LIN {X 0,Y 360.28,Z 379.159,A -85,B 0,C 180,E1 -13217.608,E2 -13217.608} C_VEL
LIN {X 0,Y 360.477,Z 375.778,A -85,B 0,C 180,E1 -13219.893,E2 -13219.893} C_VEL
LIN {X 0,Y 360.757,Z 372.266,A -85,B 0,C 180,E1 -13221.597,E2 -13221.597} C_VEL
LIN {X 0,Y 361.143,Z 367.827,A -85,B 0,C 180,E1 -13223.293,E2 -13223.293} C_VEL
LIN {X 0,Y 361.709,Z 361.416,A -85,B 0,C 180,E1 -13225.262,E2 -13225.262} C_VEL
LIN {X 0,Y 362.596,Z 353.445,A -85,B 0,C 180,E1 -13227.221,E2 -13227.221} C_VEL
LIN {X 0,Y 363.549,Z 345.118,A -85,B 0,C 180,E1 -13228.891,E2 -13228.891} C_VEL
LIN {X 0,Y 364.702,Z 335.103,A -85,B 0,C 180,E1 -13230.55,E2 -13230.55} C_VEL
LIN {X 0,Y 365.932,Z 324.301,A -85,B 0,C 180,E1 -13232.018,E2 -13232.018} C_VEL
LIN {X 0,Y 367.02,Z 312.884,A -85,B 0,C 180,E1 -13233.292,E2 -13233.292} C_VEL
LIN {X 0,Y 368.264,Z 300.783,A -85,B 0,C 180,E1 -13234.376,E2 -13234.376} C_VEL
LIN {X 0,Y 369.232,Z 287.496,A -85,B 0,C 180,E1 -13235.323,E2 -13235.323} C_VEL
LIN {X 0,Y 370.079,Z 273.64,A -85,B 0,C 180,E1 -13236.062,E2 -13236.062} C_VEL
LIN {X 0,Y 370.646,Z 259.224,A -85,B 0,C 180,E1 -13236.599,E2 -13236.599} C_VEL
LIN {X 0,Y 371.262,Z 235.703,A -85,B 0,C 180,E1 -13237.1,E2 -13237.1} C_VEL
LIN {X 0,Y 372.051,Z 196.143,A -85,B 0,C 180,E1 -13237.865,E2 -13237.865} C_VEL
LIN {X 0,Y 371.527,Z 190.322,A -85,B 0,C 180,E1 -13238.014,E2 -13238.014} C_VEL
LIN {X 0,Y 366.374,Z 171.636,A -85,B 0,C 180,E1 -13238.703,E2 -13238.703} C_VEL
LIN {X 0,Y 366.023,Z 165.818,A -85,B 0,C 180,E1 -13238.845,E2 -13238.845} C_VEL
LIN {X 0,Y 366.284,Z 150.787,A -85,B 0,C 180,E1 -13239.144,E2 -13239.144} C_VEL
LIN {X 0,Y 363.95,Z 139.954,A -85,B 0,C 180,E1 -13239.517,E2 -13239.517} C_VEL
LIN {X 0,Y 356.742,Z 120.401,A -85,B 0,C 180,E1 -13240.412,E2 -13240.412} C_VEL
LIN {X 0,Y 354.92,Z 111.908,A -85,B 0,C 180,E1 -13242.725,E2 -13242.725} C_VEL
LIN {X 0,Y 354.909,Z 111.899,A -85,B 0,C 180,E1 -13244.916,E2 -13244.916} C_VEL
LIN {X 0,Y 354.881,Z 111.901,A -85,B 0,C 180,E1 -13248.471,E2 -13248.471} C_VEL
LIN {X 0,Y 354.856,Z 111.905,A -85,B 0,C 180,E1 -13252.103,E2 -13252.103} C_VEL
LIN {X 0,Y 354.865,Z 111.905,A -85,B 0,C 180,E1 -13255.828,E2 -13255.828} C_VEL
LIN {X 0,Y 354.82,Z 111.911,A -85,B 0,C 180,E1 -13259.68,E2 -13259.68} C_VEL
LIN {X 0,Y 354.794,Z 111.913,A -85,B 0,C 180,E1 -13263.709,E2 -13263.709} C_VEL
LIN {X 0,Y 354.85,Z 111.906,A -85,B 0,C 180,E1 -13267.615,E2 -13267.615} C_VEL
LIN {X 0,Y 354.855,Z 111.907,A -85,B 0,C 180,E1 -13271.192,E2 -13271.192} C_VEL
LIN {X 0,Y 354.863,Z 111.907,A -85,B 0,C 180,E1 -13274.53,E2 -13274.53} C_VEL
LIN {X 0,Y 354.812,Z 111.91,A -85,B 0,C 180,E1 -13277.672,E2 -13277.672} C_VEL
LIN {X 0,Y 354.809,Z 111.915,A -85,B 0,C 180,E1 -13280.672,E2 -13280.672} C_VEL
LIN {X 0,Y 354.795,Z 111.916,A -85,B 0,C 180,E1 -13284.304,E2 -13284.304} C_VEL
LIN {X 0,Y 354.773,Z 111.915,A -85,B 0,C 180,E1 -13287.671,E2 -13287.671} C_VEL
LIN {X 0,Y 354.845,Z 111.908,A -85,B 0,C 180,E1 -13290.624,E2 -13290.624} C_VEL
LIN {X 0,Y 354.879,Z 111.907,A -85,B 0,C 180,E1 -13294.176,E2 -13294.176} C_VEL
LIN {X 0,Y 354.871,Z 111.907,A -85,B 0,C 180,E1 -13297.901,E2 -13297.901} C_VEL
LIN {X 0,Y 354.904,Z 111.904,A -85,B 0,C 180,E1 -13301.895,E2 -13301.895} C_VEL
LIN {X 0,Y 354.926,Z 111.9,A -85,B 0,C 180,E1 -13305.984,E2 -13305.984} C_VEL
LIN {X 0,Y 354.967,Z 111.896,A -85,B 0,C 180,E1 -13309.74,E2 -13309.74} C_VEL
LIN {X 0,Y 355.1,Z 111.875,A -85,B 0,C 180,E1 -13312.041,E2 -13312.041} C_VEL
LIN {X 0,Y 355.081,Z 111.876,A -85,B 0,C 180,E1 -13314.324,E2 -13314.324} C_VEL
LIN {X 0,Y 355.235,Z 111.86,A -85,B 0,C 180,E1 -13317.736,E2 -13317.736} C_VEL
LIN {X 0,Y 355.388,Z 111.839,A -85,B 0,C 180,E1 -13320.004,E2 -13320.004} C_VEL
LIN {X 0,Y 355.236,Z 111.857,A -85,B 0,C 180,E1 -13322.271,E2 -13322.271} C_VEL
LIN {X 0,Y 355.13,Z 111.873,A -85,B 0,C 180,E1 -13326.823,E2 -13326.823} C_VEL
LIN {X 0,Y 355.007,Z 111.891,A -85,B 0,C 180,E1 -13329.116,E2 -13329.116} C_VEL
LIN {X 0,Y 354.914,Z 111.899,A -85,B 0,C 180,E1 -13332.584,E2 -13332.584} C_VEL
LIN {X 0,Y 354.884,Z 111.901,A -85,B 0,C 180,E1 -13336.1,E2 -13336.1} C_VEL
LIN {X 0,Y 354.902,Z 111.902,A -85,B 0,C 180,E1 -13338.475,E2 -13338.475} C_VEL
LIN {X 0,Y 354.831,Z 111.909,A -85,B 0,C 180,E1 -13342.109,E2 -13342.109} C_VEL
LIN {X 0,Y 354.897,Z 111.9,A -85,B 0,C 180,E1 -13345.831,E2 -13345.831} C_VEL
LIN {X 0,Y 354.852,Z 111.905,A -85,B 0,C 180,E1 -13349.682,E2 -13349.682} C_VEL
LIN {X 0,Y 354.805,Z 111.912,A -85,B 0,C 180,E1 -13353.705,E2 -13353.705} C_VEL
LIN {X 0,Y 354.798,Z 111.915,A -85,B 0,C 180,E1 -13356.463,E2 -13356.463} C_VEL
LIN {X 0,Y 354.825,Z 111.909,A -85,B 0,C 180,E1 -13359.427,E2 -13359.427} C_VEL
LIN {X 0,Y 354.789,Z 111.913,A -85,B 0,C 180,E1 -13362.87,E2 -13362.87} C_VEL
LIN {X 0,Y 354.769,Z 111.919,A -85,B 0,C 180,E1 -13366.106,E2 -13366.106} C_VEL
LIN {X 0,Y 354.789,Z 111.913,A -85,B 0,C 180,E1 -13369.182,E2 -13369.182} C_VEL
LIN {X 0,Y 354.809,Z 111.911,A -85,B 0,C 180,E1 -13372.406,E2 -13372.406} C_VEL
LIN {X 0,Y 354.815,Z 111.91,A -85,B 0,C 180,E1 -13374.943,E2 -13374.943} C_VEL
LIN {X 0,Y 354.842,Z 111.993,A -85,B 0,C 180,E1 -13377.708,E2 -13377.708} C_VEL
LIN {X 0,Y 357.811,Z 125.266,A -85,B 0,C 180,E1 -13380.916,E2 -13380.916} C_VEL
LIN {X 0,Y 359.778,Z 135.593,A -85,B 0,C 180,E1 -13383.304,E2 -13383.304} C_VEL
LIN {X 0,Y 359.646,Z 137.884,A -85,B 0,C 180,E1 -13383.792,E2 -13383.792} C_VEL
LIN {X 0,Y 365.98,Z 177.278,A -85,B 0,C 180,E1 -13385.03,E2 -13385.03} C_VEL
LIN {X 0,Y 363.987,Z 275.483,A -85,B 0,C 180,E1 -13386.985,E2 -13386.985} C_VEL
LIN {X 0,Y 363.267,Z 289.582,A -85,B 0,C 180,E1 -13387.463,E2 -13387.463} C_VEL
LIN {X 0,Y 362.303,Z 303.328,A -85,B 0,C 180,E1 -13388.15,E2 -13388.15} C_VEL
LIN {X 0,Y 361.223,Z 315.883,A -85,B 0,C 180,E1 -13388.988,E2 -13388.988} C_VEL
LIN {X 0,Y 360.036,Z 328.122,A -85,B 0,C 180,E1 -13390.027,E2 -13390.027} C_VEL
LIN {X 0,Y 358.739,Z 340.084,A -85,B 0,C 180,E1 -13391.291,E2 -13391.291} C_VEL
LIN {X 0,Y 357.568,Z 350.013,A -85,B 0,C 180,E1 -13392.56,E2 -13392.56} C_VEL
LIN {X 0,Y 356.484,Z 359.316,A -85,B 0,C 180,E1 -13393.98,E2 -13393.98} C_VEL
LIN {X 0,Y 355.424,Z 369.309,A -85,B 0,C 180,E1 -13395.837,E2 -13395.837} C_VEL
LIN {X 0,Y 354.616,Z 377.497,A -85,B 0,C 180,E1 -13397.701,E2 -13397.701} C_VEL
LIN {X 0,Y 353.863,Z 384.642,A -85,B 0,C 180,E1 -13399.705,E2 -13399.705} C_VEL
LIN {X 0,Y 353.574,Z 389.609,A -85,B 0,C 180,E1 -13401.428,E2 -13401.428} C_VEL
LIN {X 0,Y 353.325,Z 393.615,A -85,B 0,C 180,E1 -13403.147,E2 -13403.147} C_VEL
LIN {X 0,Y 353.231,Z 397.552,A -85,B 0,C 180,E1 -13405.437,E2 -13405.437} C_VEL
LIN {X 0,Y 353.173,Z 400.031,A -85,B 0,C 180,E1 -13407.721,E2 -13407.721} C_VEL
LIN {X 0,Y 353.266,Z 401.147,A -85,B 0,C 180,E1 -13410.002,E2 -13410.002} C_VEL
LIN {X 0,Y 353.169,Z 400.916,A -85,B 0,C 180,E1 -13412.283,E2 -13412.283} C_VEL
LIN {X 0,Y 353.24,Z 399.355,A -85,B 0,C 180,E1 -13414.566,E2 -13414.566} C_VEL
LIN {X 0,Y 353.403,Z 396.435,A -85,B 0,C 180,E1 -13416.854,E2 -13416.854} C_VEL
LIN {X 0,Y 353.783,Z 392.087,A -85,B 0,C 180,E1 -13419.146,E2 -13419.146} C_VEL
LIN {X 0,Y 354.433,Z 386.192,A -85,B 0,C 180,E1 -13421.438,E2 -13421.438} C_VEL
LIN {X 0,Y 355.535,Z 379.584,A -85,B 0,C 180,E1 -13423.432,E2 -13423.432} C_VEL
LIN {X 0,Y 356.689,Z 371.416,A -85,B 0,C 180,E1 -13425.427,E2 -13425.427} C_VEL
LIN {X 0,Y 358.106,Z 362.903,A -85,B 0,C 180,E1 -13427.122,E2 -13427.122} C_VEL
LIN {X 0,Y 359.813,Z 352.629,A -85,B 0,C 180,E1 -13428.803,E2 -13428.803} C_VEL
LIN {X 0,Y 361.692,Z 341.173,A -85,B 0,C 180,E1 -13430.325,E2 -13430.325} C_VEL
LIN {X 0,Y 363.54,Z 328.705,A -85,B 0,C 180,E1 -13431.666,E2 -13431.666} C_VEL
LIN {X 0,Y 365.24,Z 315.605,A -85,B 0,C 180,E1 -13432.785,E2 -13432.785} C_VEL
LIN {X 0,Y 366.662,Z 302.384,A -85,B 0,C 180,E1 -13433.662,E2 -13433.662} C_VEL
LIN {X 0,Y 368.012,Z 287.946,A -85,B 0,C 180,E1 -13434.356,E2 -13434.356} C_VEL
LIN {X 0,Y 368.924,Z 273.358,A -85,B 0,C 180,E1 -13434.817,E2 -13434.817} C_VEL
LIN {X 0,Y 371.332,Z 177.638,A -85,B 0,C 180,E1 -13436.751,E2 -13436.751} C_VEL
LIN {X 0,Y 366.862,Z 154.52,A -85,B 0,C 180,E1 -13437.693,E2 -13437.693} C_VEL
LIN {X 0,Y 364.291,Z 144.347,A -85,B 0,C 180,E1 -13438.178,E2 -13438.178} C_VEL
LIN {X 0,Y 361.13,Z 137.187,A -85,B 0,C 180,E1 -13438.682,E2 -13438.682} C_VEL
LIN {X 0,Y 358.951,Z 127.411,A -85,B 0,C 180,E1 -13441.256,E2 -13441.256} C_VEL
LIN {X 0,Y 356.041,Z 116.351,A -85,B 0,C 180,E1 -13444.371,E2 -13444.371} C_VEL
LIN {X 0,Y 354.85,Z 111.912,A -85,B 0,C 180,E1 -13445.702,E2 -13445.702} C_VEL
LIN {X 0,Y 354.814,Z 111.911,A -85,B 0,C 180,E1 -13449.418,E2 -13449.418} C_VEL
LIN {X 0,Y 354.801,Z 111.913,A -85,B 0,C 180,E1 -13452.866,E2 -13452.866} C_VEL
LIN {X 0,Y 354.782,Z 111.92,A -85,B 0,C 180,E1 -13456.103,E2 -13456.103} C_VEL
LIN {X 0,Y 354.797,Z 111.895,A -85,B 0,C 180,E1 -13459.177,E2 -13459.177} C_VEL
LIN {X 0,Y 354.815,Z 111.908,A -85,B 0,C 180,E1 -13462.403,E2 -13462.403} C_VEL
LIN {X 0,Y 354.823,Z 111.911,A -85,B 0,C 180,E1 -13464.939,E2 -13464.939} C_VEL
LIN {X 0,Y 354.808,Z 111.909,A -85,B 0,C 180,E1 -13468.404,E2 -13468.404} C_VEL
LIN {X 0,Y 354.817,Z 111.907,A -85,B 0,C 180,E1 -13471.613,E2 -13471.613} C_VEL
LIN {X 0,Y 354.865,Z 111.899,A -85,B 0,C 180,E1 -13475.421,E2 -13475.421} C_VEL
LIN {X 0,Y 354.841,Z 111.903,A -85,B 0,C 180,E1 -13479.111,E2 -13479.111} C_VEL
LIN {X 0,Y 354.912,Z 111.899,A -85,B 0,C 180,E1 -13482.717,E2 -13482.717} C_VEL
LIN {X 0,Y 354.964,Z 111.895,A -85,B 0,C 180,E1 -13486.252,E2 -13486.252} C_VEL
LIN {X 0,Y 354.967,Z 111.891,A -85,B 0,C 180,E1 -13489.732,E2 -13489.732} C_VEL
LIN {X 0,Y 355.099,Z 111.872,A -85,B 0,C 180,E1 -13493.177,E2 -13493.177} C_VEL
LIN {X 0,Y 355.242,Z 111.852,A -85,B 0,C 180,E1 -13497.729,E2 -13497.729} C_VEL
LIN {X 0,Y 355.36,Z 111.843,A -85,B 0,C 180,E1 -13499.996,E2 -13499.996} C_VEL
LIN {X 0,Y 355.247,Z 111.856,A -85,B 0,C 180,E1 -13502.264,E2 -13502.264} C_VEL
LIN {X 0,Y 355.104,Z 111.875,A -85,B 0,C 180,E1 -13506.816,E2 -13506.816} C_VEL
LIN {X 0,Y 354.959,Z 111.892,A -85,B 0,C 180,E1 -13510.26,E2 -13510.26} C_VEL
LIN {X 0,Y 354.945,Z 111.894,A -85,B 0,C 180,E1 -13514.014,E2 -13514.014} C_VEL
LIN {X 0,Y 354.922,Z 111.899,A -85,B 0,C 180,E1 -13518.104,E2 -13518.104} C_VEL
LIN {X 0,Y 354.827,Z 111.91,A -85,B 0,C 180,E1 -13522.102,E2 -13522.102} C_VEL
LIN {X 0,Y 354.892,Z 111.898,A -85,B 0,C 180,E1 -13525.823,E2 -13525.823} C_VEL
LIN {X 0,Y 354.8,Z 111.896,A -85,B 0,C 180,E1 -13529.678,E2 -13529.678} C_VEL
LIN {X 0,Y 354.804,Z 111.903,A -85,B 0,C 180,E1 -13533.679,E2 -13533.679} C_VEL
LIN {X 0,Y 354.786,Z 111.919,A -85,B 0,C 180,E1 -13536.455,E2 -13536.455} C_VEL
LIN {X 0,Y 354.811,Z 111.916,A -85,B 0,C 180,E1 -13539.419,E2 -13539.419} C_VEL
LIN {X 0,Y 354.779,Z 112.029,A -85,B 0,C 180,E1 -13542.094,E2 -13542.094} C_VEL
LIN {X 0,Y 357.266,Z 121.425,A -85,B 0,C 180,E1 -13544.98,E2 -13544.98} C_VEL
LIN {X 0,Y 367.344,Z 141.773,A -85,B 0,C 180,E1 -13546.486,E2 -13546.486} C_VEL
LIN {X 0,Y 371.616,Z 152.058,A -85,B 0,C 180,E1 -13547.126,E2 -13547.126} C_VEL
LIN {X 0,Y 371.984,Z 155.184,A -85,B 0,C 180,E1 -13547.23,E2 -13547.23} C_VEL
LIN {X 0,Y 369.169,Z 257.932,A -85,B 0,C 180,E1 -13549.303,E2 -13549.303} C_VEL
LIN {X 0,Y 368.327,Z 272.35,A -85,B 0,C 180,E1 -13549.815,E2 -13549.815} C_VEL
LIN {X 0,Y 367.121,Z 286.785,A -85,B 0,C 180,E1 -13550.569,E2 -13550.569} C_VEL
LIN {X 0,Y 365.711,Z 300.307,A -85,B 0,C 180,E1 -13551.524,E2 -13551.524} C_VEL
LIN {X 0,Y 364.152,Z 312.611,A -85,B 0,C 180,E1 -13552.634,E2 -13552.634} C_VEL
LIN {X 0,Y 362.478,Z 324.097,A -85,B 0,C 180,E1 -13553.917,E2 -13553.917} C_VEL
LIN {X 0,Y 360.851,Z 334.55,A -85,B 0,C 180,E1 -13555.345,E2 -13555.345} C_VEL
LIN {X 0,Y 359.349,Z 343.369,A -85,B 0,C 180,E1 -13556.795,E2 -13556.795} C_VEL
LIN {X 0,Y 357.753,Z 352.616,A -85,B 0,C 180,E1 -13558.627,E2 -13558.627} C_VEL
LIN {X 0,Y 356.399,Z 360.167,A -85,B 0,C 180,E1 -13560.461,E2 -13560.461} C_VEL
LIN {X 0,Y 355.416,Z 366.333,A -85,B 0,C 180,E1 -13562.308,E2 -13562.308} C_VEL
LIN {X 0,Y 354.591,Z 371.3,A -85,B 0,C 180,E1 -13564.147,E2 -13564.147} C_VEL
LIN {X 0,Y 354.04,Z 375.121,A -85,B 0,C 180,E1 -13565.929,E2 -13565.929} C_VEL
LIN {X 0,Y 353.596,Z 378.199,A -85,B 0,C 180,E1 -13567.811,E2 -13567.811} C_VEL
LIN {X 0,Y 353.224,Z 380.722,A -85,B 0,C 180,E1 -13570.228,E2 -13570.228} C_VEL
LIN {X 0,Y 353.081,Z 381.77,A -85,B 0,C 180,E1 -13572.627,E2 -13572.627} C_VEL
LIN {X 0,Y 353.002,Z 381.395,A -85,B 0,C 180,E1 -13574.998,E2 -13574.998} C_VEL
LIN {X 0,Y 353.166,Z 379.613,A -85,B 0,C 180,E1 -13577.354,E2 -13577.354} C_VEL
LIN {X 0,Y 353.349,Z 376.424,A -85,B 0,C 180,E1 -13579.686,E2 -13579.686} C_VEL
LIN {X 0,Y 353.639,Z 373.009,A -85,B 0,C 180,E1 -13581.427,E2 -13581.427} C_VEL
LIN {X 0,Y 354.195,Z 367.1,A -85,B 0,C 180,E1 -13583.733,E2 -13583.733} C_VEL
LIN {X 0,Y 354.834,Z 360.46,A -85,B 0,C 180,E1 -13585.739,E2 -13585.739} C_VEL
LIN {X 0,Y 355.776,Z 352.193,A -85,B 0,C 180,E1 -13587.734,E2 -13587.734} C_VEL
LIN {X 0,Y 356.804,Z 343.568,A -85,B 0,C 180,E1 -13589.434,E2 -13589.434} C_VEL
LIN {X 0,Y 358.02,Z 333.131,A -85,B 0,C 180,E1 -13591.123,E2 -13591.123} C_VEL
LIN {X 0,Y 359.353,Z 321.46,A -85,B 0,C 180,E1 -13592.661,E2 -13592.661} C_VEL
LIN {X 0,Y 360.595,Z 309.782,A -85,B 0,C 180,E1 -13593.91,E2 -13593.91} C_VEL
LIN {X 0,Y 361.772,Z 296.951,A -85,B 0,C 180,E1 -13595.014,E2 -13595.014} C_VEL
LIN {X 0,Y 362.808,Z 283.611,A -85,B 0,C 180,E1 -13595.905,E2 -13595.905} C_VEL
LIN {X 0,Y 363.558,Z 269.855,A -85,B 0,C 180,E1 -13596.589,E2 -13596.589} C_VEL
LIN {X 0,Y 364.059,Z 255.517,A -85,B 0,C 180,E1 -13597.067,E2 -13597.067} C_VEL
LIN {X 0,Y 366.023,Z 165.818,A -85,B 0,C 180,E1 -13598.845,E2 -13598.845} C_VEL
LIN {X 0,Y 365.619,Z 159.993,A -85,B 0,C 180,E1 -13598.992,E2 -13598.992} C_VEL
LIN {X 0,Y 364.039,Z 154.409,A -85,B 0,C 180,E1 -13599.207,E2 -13599.207} C_VEL
LIN {X 0,Y 359.047,Z 143.816,A -85,B 0,C 180,E1 -13599.745,E2 -13599.745} C_VEL
LIN {X 0,Y 355.643,Z 136.727,A -85,B 0,C 180,E1 -13600.119,E2 -13600.119} C_VEL
LIN {X 0,Y 349.585,Z 120.631,A -85,B 0,C 180,E1 -13600.89,E2 -13600.89} C_VEL
LIN {X 0,Y 347.909,Z 112.78,A -85,B 0,C 180,E1 -13603.06,E2 -13603.06} C_VEL
LIN {X 0,Y 347.824,Z 112.782,A -85,B 0,C 180,E1 -13606.43,E2 -13606.43} C_VEL
LIN {X 0,Y 347.831,Z 112.781,A -85,B 0,C 180,E1 -13608.86,E2 -13608.86} C_VEL
LIN {X 0,Y 347.776,Z 112.787,A -85,B 0,C 180,E1 -13612.577,E2 -13612.577} C_VEL
LIN {X 0,Y 347.786,Z 112.789,A -85,B 0,C 180,E1 -13615.108,E2 -13615.108} C_VEL
LIN {X 0,Y 347.777,Z 112.788,A -85,B 0,C 180,E1 -13617.695,E2 -13617.695} C_VEL
LIN {X 0,Y 347.736,Z 112.791,A -85,B 0,C 180,E1 -13620.347,E2 -13620.347} C_VEL
LIN {X 0,Y 347.731,Z 112.792,A -85,B 0,C 180,E1 -13624.049,E2 -13624.049} C_VEL
LIN {X 0,Y 347.794,Z 112.787,A -85,B 0,C 180,E1 -13627.314,E2 -13627.314} C_VEL
LIN {X 0,Y 347.787,Z 112.786,A -85,B 0,C 180,E1 -13630.287,E2 -13630.287} C_VEL
LIN {X 0,Y 347.79,Z 112.784,A -85,B 0,C 180,E1 -13633.395,E2 -13633.395} C_VEL
LIN {X 0,Y 347.789,Z 112.79,A -85,B 0,C 180,E1 -13636.672,E2 -13636.672} C_VEL
LIN {X 0,Y 347.757,Z 112.79,A -85,B 0,C 180,E1 -13640.168,E2 -13640.168} C_VEL
LIN {X 0,Y 347.763,Z 112.79,A -85,B 0,C 180,E1 -13644.128,E2 -13644.128} C_VEL
LIN {X 0,Y 347.74,Z 112.796,A -85,B 0,C 180,E1 -13648.306,E2 -13648.306} C_VEL
LIN {X 0,Y 347.783,Z 112.784,A -85,B 0,C 180,E1 -13650.993,E2 -13650.993} C_VEL
LIN {X 0,Y 347.81,Z 112.782,A -85,B 0,C 180,E1 -13653.611,E2 -13653.611} C_VEL
LIN {X 0,Y 347.797,Z 112.789,A -85,B 0,C 180,E1 -13656.168,E2 -13656.168} C_VEL
LIN {X 0,Y 347.825,Z 112.785,A -85,B 0,C 180,E1 -13659.915,E2 -13659.915} C_VEL
LIN {X 0,Y 347.849,Z 112.779,A -85,B 0,C 180,E1 -13662.363,E2 -13662.363} C_VEL
LIN {X 0,Y 347.88,Z 112.777,A -85,B 0,C 180,E1 -13665.975,E2 -13665.975} C_VEL
LIN {X 0,Y 347.918,Z 112.773,A -85,B 0,C 180,E1 -13669.53,E2 -13669.53} C_VEL
LIN {X 0,Y 348.06,Z 112.753,A -85,B 0,C 180,E1 -13671.879,E2 -13671.879} C_VEL
LIN {X 0,Y 348.056,Z 112.75,A -85,B 0,C 180,E1 -13674.21,E2 -13674.21} C_VEL
LIN {X 0,Y 348.198,Z 112.737,A -85,B 0,C 180,E1 -13677.69,E2 -13677.69} C_VEL
LIN {X 0,Y 348.358,Z 112.714,A -85,B 0,C 180,E1 -13680.004,E2 -13680.004} C_VEL
LIN {X 0,Y 348.199,Z 112.733,A -85,B 0,C 180,E1 -13682.317,E2 -13682.317} C_VEL
LIN {X 0,Y 348.098,Z 112.749,A -85,B 0,C 180,E1 -13686.961,E2 -13686.961} C_VEL
LIN {X 0,Y 347.96,Z 112.767,A -85,B 0,C 180,E1 -13689.302,E2 -13689.302} C_VEL
LIN {X 0,Y 347.883,Z 112.778,A -85,B 0,C 180,E1 -13692.843,E2 -13692.843} C_VEL
LIN {X 0,Y 347.834,Z 112.781,A -85,B 0,C 180,E1 -13696.435,E2 -13696.435} C_VEL
LIN {X 0,Y 347.851,Z 112.782,A -85,B 0,C 180,E1 -13698.864,E2 -13698.864} C_VEL
LIN {X 0,Y 347.771,Z 112.792,A -85,B 0,C 180,E1 -13702.583,E2 -13702.583} C_VEL
LIN {X 0,Y 347.809,Z 112.783,A -85,B 0,C 180,E1 -13705.112,E2 -13705.112} C_VEL
LIN {X 0,Y 347.809,Z 112.782,A -85,B 0,C 180,E1 -13707.697,E2 -13707.697} C_VEL
LIN {X 0,Y 347.762,Z 112.793,A -85,B 0,C 180,E1 -13710.35,E2 -13710.35} C_VEL
LIN {X 0,Y 347.744,Z 112.794,A -85,B 0,C 180,E1 -13714.467,E2 -13714.467} C_VEL
LIN {X 0,Y 347.773,Z 112.791,A -85,B 0,C 180,E1 -13717.992,E2 -13717.992} C_VEL
LIN {X 0,Y 347.752,Z 112.793,A -85,B 0,C 180,E1 -13721.833,E2 -13721.833} C_VEL
LIN {X 0,Y 347.707,Z 112.795,A -85,B 0,C 180,E1 -13725.03,E2 -13725.03} C_VEL
LIN {X 0,Y 347.752,Z 112.79,A -85,B 0,C 180,E1 -13728.4,E2 -13728.4} C_VEL
LIN {X 0,Y 347.775,Z 112.79,A -85,B 0,C 180,E1 -13732.015,E2 -13732.015} C_VEL
LIN {X 0,Y 347.748,Z 112.796,A -85,B 0,C 180,E1 -13735.539,E2 -13735.539} C_VEL
LIN {X 0,Y 347.767,Z 112.852,A -85,B 0,C 180,E1 -13737.33,E2 -13737.33} C_VEL
LIN {X 0,Y 350.758,Z 126.06,A -85,B 0,C 180,E1 -13740.603,E2 -13740.603} C_VEL
LIN {X 0,Y 352.793,Z 136.523,A -85,B 0,C 180,E1 -13743.078,E2 -13743.078} C_VEL
LIN {X 0,Y 352.875,Z 138.029,A -85,B 0,C 180,E1 -13743.362,E2 -13743.362} C_VEL
LIN {X 0,Y 359.356,Z 177.632,A -85,B 0,C 180,E1 -13744.635,E2 -13744.635} C_VEL
LIN {X 0,Y 357.293,Z 275.037,A -85,B 0,C 180,E1 -13746.605,E2 -13746.605} C_VEL
LIN {X 0,Y 356.54,Z 289.244,A -85,B 0,C 180,E1 -13747.091,E2 -13747.091} C_VEL
LIN {X 0,Y 355.572,Z 303.032,A -85,B 0,C 180,E1 -13747.791,E2 -13747.791} C_VEL
LIN {X 0,Y 354.382,Z 316.303,A -85,B 0,C 180,E1 -13748.698,E2 -13748.698} C_VEL
LIN {X 0,Y 353.124,Z 328.581,A -85,B 0,C 180,E1 -13749.771,E2 -13749.771} C_VEL
LIN {X 0,Y 351.814,Z 340.431,A -85,B 0,C 180,E1 -13751.059,E2 -13751.059} C_VEL
LIN {X 0,Y 350.475,Z 351.256,A -85,B 0,C 180,E1 -13752.497,E2 -13752.497} C_VEL
LIN {X 0,Y 349.191,Z 361.973,A -85,B 0,C 180,E1 -13754.236,E2 -13754.236} C_VEL
LIN {X 0,Y 348.288,Z 370.812,A -85,B 0,C 180,E1 -13755.989,E2 -13755.989} C_VEL
LIN {X 0,Y 347.355,Z 379.259,A -85,B 0,C 180,E1 -13758.032,E2 -13758.032} C_VEL
LIN {X 0,Y 346.697,Z 386.022,A -85,B 0,C 180,E1 -13760.08,E2 -13760.08} C_VEL
LIN {X 0,Y 346.41,Z 390.67,A -85,B 0,C 180,E1 -13761.837,E2 -13761.837} C_VEL
LIN {X 0,Y 346.135,Z 395.453,A -85,B 0,C 180,E1 -13764.175,E2 -13764.175} C_VEL
LIN {X 0,Y 346.13,Z 398.7,A -85,B 0,C 180,E1 -13766.509,E2 -13766.509} C_VEL
LIN {X 0,Y 346.121,Z 400.531,A -85,B 0,C 180,E1 -13768.838,E2 -13768.838} C_VEL
LIN {X 0,Y 346.169,Z 400.94,A -85,B 0,C 180,E1 -13770.002,E2 -13770.002} C_VEL
LIN {X 0,Y 346.08,Z 400.75,A -85,B 0,C 180,E1 -13772.329,E2 -13772.329} C_VEL
LIN {X 0,Y 346.14,Z 399.231,A -85,B 0,C 180,E1 -13774.66,E2 -13774.66} C_VEL
LIN {X 0,Y 346.328,Z 396.357,A -85,B 0,C 180,E1 -13776.995,E2 -13776.995} C_VEL
LIN {X 0,Y 346.731,Z 392.055,A -85,B 0,C 180,E1 -13779.334,E2 -13779.334} C_VEL
LIN {X 0,Y 347.446,Z 386.209,A -85,B 0,C 180,E1 -13781.672,E2 -13781.672} C_VEL
LIN {X 0,Y 348.581,Z 379.654,A -85,B 0,C 180,E1 -13783.705,E2 -13783.705} C_VEL
LIN {X 0,Y 349.825,Z 371.559,A -85,B 0,C 180,E1 -13785.738,E2 -13785.738} C_VEL
LIN {X 0,Y 351.325,Z 363.111,A -85,B 0,C 180,E1 -13787.463,E2 -13787.463} C_VEL
LIN {X 0,Y 353.117,Z 352.958,A -85,B 0,C 180,E1 -13789.173,E2 -13789.173} C_VEL
LIN {X 0,Y 355.066,Z 341.625,A -85,B 0,C 180,E1 -13790.722,E2 -13790.722} C_VEL
LIN {X 0,Y 356.849,Z 330.395,A -85,B 0,C 180,E1 -13791.976,E2 -13791.976} C_VEL
LIN {X 0,Y 358.516,Z 318.17,A -85,B 0,C 180,E1 -13793.084,E2 -13793.084} C_VEL
LIN {X 0,Y 360.133,Z 304.59,A -85,B 0,C 180,E1 -13794.042,E2 -13794.042} C_VEL
LIN {X 0,Y 361.473,Z 291.074,A -85,B 0,C 180,E1 -13794.749,E2 -13794.749} C_VEL
LIN {X 0,Y 362.524,Z 277.279,A -85,B 0,C 180,E1 -13795.247,E2 -13795.247} C_VEL
LIN {X 0,Y 363.289,Z 252.132,A -85,B 0,C 180,E1 -13795.804,E2 -13795.804} C_VEL
LIN {X 0,Y 365.226,Z 178.802,A -85,B 0,C 180,E1 -13797.295,E2 -13797.295} C_VEL
LIN {X 0,Y 360.808,Z 155.911,A -85,B 0,C 180,E1 -13798.257,E2 -13798.257} C_VEL
LIN {X 0,Y 358.729,Z 147.618,A -85,B 0,C 180,E1 -13798.665,E2 -13798.665} C_VEL
LIN {X 0,Y 353.974,Z 136.861,A -85,B 0,C 180,E1 -13799.462,E2 -13799.462} C_VEL
LIN {X 0,Y 351.325,Z 125.937,A -85,B 0,C 180,E1 -13802.47,E2 -13802.47} C_VEL
LIN {X 0,Y 348.62,Z 115.935,A -85,B 0,C 180,E1 -13805.423,E2 -13805.423} C_VEL
LIN {X 0,Y 347.773,Z 112.79,A -85,B 0,C 180,E1 -13806.43,E2 -13806.43} C_VEL
LIN {X 0,Y 347.742,Z 112.786,A -85,B 0,C 180,E1 -13809.822,E2 -13809.822} C_VEL
LIN {X 0,Y 347.738,Z 112.793,A -85,B 0,C 180,E1 -13813.408,E2 -13813.408} C_VEL
LIN {X 0,Y 347.74,Z 112.795,A -85,B 0,C 180,E1 -13816.686,E2 -13816.686} C_VEL
LIN {X 0,Y 347.743,Z 112.785,A -85,B 0,C 180,E1 -13820.176,E2 -13820.176} C_VEL
LIN {X 0,Y 347.771,Z 112.784,A -85,B 0,C 180,E1 -13822.677,E2 -13822.677} C_VEL
LIN {X 0,Y 347.763,Z 112.786,A -85,B 0,C 180,E1 -13825.955,E2 -13825.955} C_VEL
LIN {X 0,Y 347.753,Z 112.79,A -85,B 0,C 180,E1 -13829.649,E2 -13829.649} C_VEL
LIN {X 0,Y 347.77,Z 112.791,A -85,B 0,C 180,E1 -13833.6,E2 -13833.6} C_VEL
LIN {X 0,Y 347.785,Z 112.778,A -85,B 0,C 180,E1 -13836.158,E2 -13836.158} C_VEL
LIN {X 0,Y 347.814,Z 112.774,A -85,B 0,C 180,E1 -13839.906,E2 -13839.906} C_VEL
LIN {X 0,Y 347.88,Z 112.777,A -85,B 0,C 180,E1 -13842.357,E2 -13842.357} C_VEL
LIN {X 0,Y 347.911,Z 112.772,A -85,B 0,C 180,E1 -13845.968,E2 -13845.968} C_VEL
LIN {X 0,Y 347.908,Z 112.77,A -85,B 0,C 180,E1 -13849.521,E2 -13849.521} C_VEL
LIN {X 0,Y 348.066,Z 112.747,A -85,B 0,C 180,E1 -13853.038,E2 -13853.038} C_VEL
LIN {X 0,Y 348.204,Z 112.728,A -85,B 0,C 180,E1 -13857.683,E2 -13857.683} C_VEL
LIN {X 0,Y 348.31,Z 112.72,A -85,B 0,C 180,E1 -13859.996,E2 -13859.996} C_VEL
LIN {X 0,Y 348.209,Z 112.732,A -85,B 0,C 180,E1 -13862.31,E2 -13862.31} C_VEL
LIN {X 0,Y 348.072,Z 112.751,A -85,B 0,C 180,E1 -13866.954,E2 -13866.954} C_VEL
LIN {X 0,Y 347.9,Z 112.773,A -85,B 0,C 180,E1 -13870.471,E2 -13870.471} C_VEL
LIN {X 0,Y 347.9,Z 112.773,A -85,B 0,C 180,E1 -13874.145,E2 -13874.145} C_VEL
LIN {X 0,Y 347.89,Z 112.775,A -85,B 0,C 180,E1 -13878.285,E2 -13878.285} C_VEL
LIN {X 0,Y 347.784,Z 112.79,A -85,B 0,C 180,E1 -13881.629,E2 -13881.629} C_VEL
LIN {X 0,Y 347.806,Z 112.787,A -85,B 0,C 180,E1 -13885.104,E2 -13885.104} C_VEL
LIN {X 0,Y 347.795,Z 112.787,A -85,B 0,C 180,E1 -13887.69,E2 -13887.69} C_VEL
LIN {X 0,Y 347.737,Z 112.777,A -85,B 0,C 180,E1 -13890.344,E2 -13890.344} C_VEL
LIN {X 0,Y 347.738,Z 112.781,A -85,B 0,C 180,E1 -13894.039,E2 -13894.039} C_VEL
LIN {X 0,Y 347.749,Z 112.785,A -85,B 0,C 180,E1 -13897.316,E2 -13897.316} C_VEL
LIN {X 0,Y 347.73,Z 112.789,A -85,B 0,C 180,E1 -13901.353,E2 -13901.353} C_VEL
LIN {X 0,Y 350.05,Z 121.553,A -85,B 0,C 180,E1 -13904.186,E2 -13904.186} C_VEL
LIN {X 0,Y 361.108,Z 143.489,A -85,B 0,C 180,E1 -13905.905,E2 -13905.905} C_VEL
LIN {X 0,Y 365.814,Z 154.641,A -85,B 0,C 180,E1 -13906.632,E2 -13906.632} C_VEL
LIN {X 0,Y 365.393,Z 174.831,A -85,B 0,C 180,E1 -13907.055,E2 -13907.055} C_VEL
LIN {X 0,Y 363.021,Z 257.317,A -85,B 0,C 180,E1 -13908.741,E2 -13908.741} C_VEL
LIN {X 0,Y 362.136,Z 272.069,A -85,B 0,C 180,E1 -13909.261,E2 -13909.261} C_VEL
LIN {X 0,Y 360.91,Z 286.391,A -85,B 0,C 180,E1 -13910.012,E2 -13910.012} C_VEL
LIN {X 0,Y 359.543,Z 299.259,A -85,B 0,C 180,E1 -13910.919,E2 -13910.919} C_VEL
LIN {X 0,Y 357.92,Z 311.436,A -85,B 0,C 180,E1 -13912.006,E2 -13912.006} C_VEL
LIN {X 0,Y 356.308,Z 322.188,A -85,B 0,C 180,E1 -13913.191,E2 -13913.191} C_VEL
LIN {X 0,Y 354.478,Z 333.398,A -85,B 0,C 180,E1 -13914.7,E2 -13914.7} C_VEL
LIN {X 0,Y 352.686,Z 343.448,A -85,B 0,C 180,E1 -13916.353,E2 -13916.353} C_VEL
LIN {X 0,Y 350.949,Z 353.014,A -85,B 0,C 180,E1 -13918.285,E2 -13918.285} C_VEL
LIN {X 0,Y 349.538,Z 360.531,A -85,B 0,C 180,E1 -13920.155,E2 -13920.155} C_VEL
LIN {X 0,Y 348.318,Z 367.567,A -85,B 0,C 180,E1 -13922.348,E2 -13922.348} C_VEL
LIN {X 0,Y 347.497,Z 372.354,A -85,B 0,C 180,E1 -13924.224,E2 -13924.224} C_VEL
LIN {X 0,Y 346.915,Z 376.06,A -85,B 0,C 180,E1 -13926.096,E2 -13926.096} C_VEL
LIN {X 0,Y 346.371,Z 379.583,A -85,B 0,C 180,E1 -13928.577,E2 -13928.577} C_VEL
LIN {X 0,Y 346.056,Z 381.521,A -85,B 0,C 180,E1 -13931.036,E2 -13931.036} C_VEL
LIN {X 0,Y 345.938,Z 381.994,A -85,B 0,C 180,E1 -13933.474,E2 -13933.474} C_VEL
LIN {X 0,Y 345.953,Z 381.055,A -85,B 0,C 180,E1 -13935.889,E2 -13935.889} C_VEL
LIN {X 0,Y 346.057,Z 380.057,A -85,B 0,C 180,E1 -13937.09,E2 -13937.09} C_VEL
LIN {X 0,Y 346.22,Z 377.009,A -85,B 0,C 180,E1 -13939.472,E2 -13939.472} C_VEL
LIN {X 0,Y 346.542,Z 373.738,A -85,B 0,C 180,E1 -13941.25,E2 -13941.25} C_VEL
LIN {X 0,Y 347.068,Z 367.943,A -85,B 0,C 180,E1 -13943.619,E2 -13943.619} C_VEL
LIN {X 0,Y 347.695,Z 361.515,A -85,B 0,C 180,E1 -13945.651,E2 -13945.651} C_VEL
LIN {X 0,Y 348.659,Z 353.476,A -85,B 0,C 180,E1 -13947.688,E2 -13947.688} C_VEL
LIN {X 0,Y 349.698,Z 345.07,A -85,B 0,C 180,E1 -13949.423,E2 -13949.423} C_VEL
LIN {X 0,Y 350.95,Z 334.954,A -85,B 0,C 180,E1 -13951.146,E2 -13951.146} C_VEL
LIN {X 0,Y 352.279,Z 323.633,A -85,B 0,C 180,E1 -13952.714,E2 -13952.714} C_VEL
LIN {X 0,Y 353.462,Z 312.405,A -85,B 0,C 180,E1 -13953.989,E2 -13953.989} C_VEL
LIN {X 0,Y 354.745,Z 300.108,A -85,B 0,C 180,E1 -13955.113,E2 -13955.113} C_VEL
LIN {X 0,Y 355.84,Z 286.493,A -85,B 0,C 180,E1 -13956.092,E2 -13956.092} C_VEL
LIN {X 0,Y 356.753,Z 272.156,A -85,B 0,C 180,E1 -13956.858,E2 -13956.858} C_VEL
LIN {X 0,Y 357.296,Z 257.985,A -85,B 0,C 180,E1 -13957.379,E2 -13957.379} C_VEL
LIN {X 0,Y 359.312,Z 172.015,A -85,B 0,C 180,E1 -13959.126,E2 -13959.126} C_VEL
LIN {X 0,Y 359.593,Z 151.462,A -85,B 0,C 180,E1 -13959.547,E2 -13959.547} C_VEL
LIN {X 0,Y 357.534,Z 142.054,A -85,B 0,C 180,E1 -13959.88,E2 -13959.88} C_VEL
LIN {X 0,Y 355.643,Z 136.727,A -85,B 0,C 180,E1 -13960.119,E2 -13960.119} C_VEL
LIN {X 0,Y 353.601,Z 133.517,A -85,B 0,C 180,E1 -13960.325,E2 -13960.325} C_VEL
LIN {X 0,Y 344.427,Z 124.942,A -85,B 0,C 180,E1 -13961.149,E2 -13961.149} C_VEL
LIN {X 0,Y 342.624,Z 121.633,A -85,B 0,C 180,E1 -13961.351,E2 -13961.351} C_VEL
LIN {X 0,Y 342.359,Z 120.679,A -85,B 0,C 180,E1 -13961.432,E2 -13961.432} C_VEL
LIN {X 0,Y 340.859,Z 113.656,A -85,B 0,C 180,E1 -13963.4,E2 -13963.4} C_VEL
LIN {X 0,Y 340.771,Z 113.661,A -85,B 0,C 180,E1 -13966.78,E2 -13966.78} C_VEL
LIN {X 0,Y 340.773,Z 113.663,A -85,B 0,C 180,E1 -13969.266,E2 -13969.266} C_VEL
LIN {X 0,Y 340.742,Z 113.665,A -85,B 0,C 180,E1 -13973.07,E2 -13973.07} C_VEL
LIN {X 0,Y 340.77,Z 113.662,A -85,B 0,C 180,E1 -13976.981,E2 -13976.981} C_VEL
LIN {X 0,Y 340.731,Z 113.664,A -85,B 0,C 180,E1 -13979.98,E2 -13979.98} C_VEL
LIN {X 0,Y 340.674,Z 113.672,A -85,B 0,C 180,E1 -13983.846,E2 -13983.846} C_VEL
LIN {X 0,Y 340.739,Z 113.666,A -85,B 0,C 180,E1 -13986.735,E2 -13986.735} C_VEL
LIN {X 0,Y 340.758,Z 113.661,A -85,B 0,C 180,E1 -13990.269,E2 -13990.269} C_VEL
LIN {X 0,Y 340.753,Z 113.659,A -85,B 0,C 180,E1 -13993.798,E2 -13993.798} C_VEL
LIN {X 0,Y 340.733,Z 113.666,A -85,B 0,C 180,E1 -13997.112,E2 -13997.112} C_VEL
LIN {X 0,Y 340.706,Z 113.669,A -85,B 0,C 180,E1 -14000.255,E2 -14000.255} C_VEL
LIN {X 0,Y 340.685,Z 113.668,A -85,B 0,C 180,E1 -14003.562,E2 -14003.562} C_VEL
LIN {X 0,Y 340.669,Z 113.675,A -85,B 0,C 180,E1 -14006.157,E2 -14006.157} C_VEL
LIN {X 0,Y 340.752,Z 113.663,A -85,B 0,C 180,E1 -14010.336,E2 -14010.336} C_VEL
LIN {X 0,Y 340.783,Z 113.656,A -85,B 0,C 180,E1 -14013.024,E2 -14013.024} C_VEL
LIN {X 0,Y 340.756,Z 113.661,A -85,B 0,C 180,E1 -14016.934,E2 -14016.934} C_VEL
LIN {X 0,Y 340.787,Z 113.657,A -85,B 0,C 180,E1 -14020.738,E2 -14020.738} C_VEL
LIN {X 0,Y 340.77,Z 113.66,A -85,B 0,C 180,E1 -14023.222,E2 -14023.222} C_VEL
LIN {X 0,Y 340.83,Z 113.651,A -85,B 0,C 180,E1 -14026.894,E2 -14026.894} C_VEL
LIN {X 0,Y 340.915,Z 113.64,A -85,B 0,C 180,E1 -14030.512,E2 -14030.512} C_VEL
LIN {X 0,Y 341.062,Z 113.621,A -85,B 0,C 180,E1 -14032.902,E2 -14032.902} C_VEL
LIN {X 0,Y 341.16,Z 113.614,A -85,B 0,C 180,E1 -14037.643,E2 -14037.643} C_VEL
LIN {X 0,Y 341.307,Z 113.593,A -85,B 0,C 180,E1 -14040.004,E2 -14040.004} C_VEL
LIN {X 0,Y 341.161,Z 113.609,A -85,B 0,C 180,E1 -14042.365,E2 -14042.365} C_VEL
LIN {X 0,Y 341.067,Z 113.626,A -85,B 0,C 180,E1 -14047.106,E2 -14047.106} C_VEL
LIN {X 0,Y 340.864,Z 113.65,A -85,B 0,C 180,E1 -14050.698,E2 -14050.698} C_VEL
LIN {X 0,Y 340.857,Z 113.649,A -85,B 0,C 180,E1 -14054.329,E2 -14054.329} C_VEL
LIN {X 0,Y 340.833,Z 113.654,A -85,B 0,C 180,E1 -14058.471,E2 -14058.471} C_VEL
LIN {X 0,Y 340.75,Z 113.662,A -85,B 0,C 180,E1 -14061.861,E2 -14061.861} C_VEL
LIN {X 0,Y 340.77,Z 113.659,A -85,B 0,C 180,E1 -14065.668,E2 -14065.668} C_VEL
LIN {X 0,Y 340.739,Z 113.666,A -85,B 0,C 180,E1 -14068.323,E2 -14068.323} C_VEL
LIN {X 0,Y 340.702,Z 113.668,A -85,B 0,C 180,E1 -14071.048,E2 -14071.048} C_VEL
LIN {X 0,Y 340.717,Z 113.665,A -85,B 0,C 180,E1 -14075.282,E2 -14075.282} C_VEL
LIN {X 0,Y 340.71,Z 113.67,A -85,B 0,C 180,E1 -14078.389,E2 -14078.389} C_VEL
LIN {X 0,Y 340.7,Z 113.673,A -85,B 0,C 180,E1 -14082.049,E2 -14082.049} C_VEL
LIN {X 0,Y 340.654,Z 113.677,A -85,B 0,C 180,E1 -14086.23,E2 -14086.23} C_VEL
LIN {X 0,Y 340.691,Z 113.674,A -85,B 0,C 180,E1 -14089.756,E2 -14089.756} C_VEL
LIN {X 0,Y 340.708,Z 113.67,A -85,B 0,C 180,E1 -14093.261,E2 -14093.261} C_VEL
LIN {X 0,Y 340.725,Z 113.808,A -85,B 0,C 180,E1 -14096.965,E2 -14096.965} C_VEL
LIN {X 0,Y 343.703,Z 126.908,A -85,B 0,C 180,E1 -14100.289,E2 -14100.289} C_VEL
LIN {X 0,Y 345.841,Z 137.723,A -85,B 0,C 180,E1 -14102.874,E2 -14102.874} C_VEL
LIN {X 0,Y 347.364,Z 145.216,A -85,B 0,C 180,E1 -14103.146,E2 -14103.146} C_VEL
LIN {X 0,Y 352.721,Z 179.215,A -85,B 0,C 180,E1 -14104.25,E2 -14104.25} C_VEL
LIN {X 0,Y 350.615,Z 274.567,A -85,B 0,C 180,E1 -14106.211,E2 -14106.211} C_VEL
LIN {X 0,Y 349.86,Z 288.913,A -85,B 0,C 180,E1 -14106.706,E2 -14106.706} C_VEL
LIN {X 0,Y 348.849,Z 302.734,A -85,B 0,C 180,E1 -14107.418,E2 -14107.418} C_VEL
LIN {X 0,Y 347.8,Z 314.538,A -85,B 0,C 180,E1 -14108.222,E2 -14108.222} C_VEL
LIN {X 0,Y 346.403,Z 327.599,A -85,B 0,C 180,E1 -14109.361,E2 -14109.361} C_VEL
LIN {X 0,Y 345.177,Z 338.398,A -85,B 0,C 180,E1 -14110.526,E2 -14110.526} C_VEL
LIN {X 0,Y 343.907,Z 348.543,A -85,B 0,C 180,E1 -14111.843,E2 -14111.843} C_VEL
LIN {X 0,Y 342.5,Z 359.678,A -85,B 0,C 180,E1 -14113.614,E2 -14113.614} C_VEL
LIN {X 0,Y 341.489,Z 368.464,A -85,B 0,C 180,E1 -14115.311,E2 -14115.311} C_VEL
LIN {X 0,Y 340.582,Z 376.496,A -85,B 0,C 180,E1 -14117.185,E2 -14117.185} C_VEL
LIN {X 0,Y 339.781,Z 383.762,A -85,B 0,C 180,E1 -14119.273,E2 -14119.273} C_VEL
LIN {X 0,Y 339.45,Z 388.837,A -85,B 0,C 180,E1 -14121.069,E2 -14121.069} C_VEL
LIN {X 0,Y 339.173,Z 392.896,A -85,B 0,C 180,E1 -14122.86,E2 -14122.86} C_VEL
LIN {X 0,Y 339.031,Z 396.954,A -85,B 0,C 180,E1 -14125.245,E2 -14125.245} C_VEL
LIN {X 0,Y 339.053,Z 398.425,A -85,B 0,C 180,E1 -14126.436,E2 -14126.436} C_VEL
LIN {X 0,Y 339.023,Z 400.302,A -85,B 0,C 180,E1 -14128.814,E2 -14128.814} C_VEL
LIN {X 0,Y 339.072,Z 400.733,A -85,B 0,C 180,E1 -14130.002,E2 -14130.002} C_VEL
LIN {X 0,Y 338.995,Z 400.586,A -85,B 0,C 180,E1 -14132.378,E2 -14132.378} C_VEL
LIN {X 0,Y 339.044,Z 399.109,A -85,B 0,C 180,E1 -14134.758,E2 -14134.758} C_VEL
LIN {X 0,Y 339.257,Z 396.279,A -85,B 0,C 180,E1 -14137.142,E2 -14137.142} C_VEL
LIN {X 0,Y 339.695,Z 392.023,A -85,B 0,C 180,E1 -14139.529,E2 -14139.529} C_VEL
LIN {X 0,Y 340.473,Z 386.226,A -85,B 0,C 180,E1 -14141.914,E2 -14141.914} C_VEL
LIN {X 0,Y 341.634,Z 379.731,A -85,B 0,C 180,E1 -14143.99,E2 -14143.99} C_VEL
LIN {X 0,Y 342.97,Z 371.71,A -85,B 0,C 180,E1 -14146.061,E2 -14146.061} C_VEL
LIN {X 0,Y 344.529,Z 363.341,A -85,B 0,C 180,E1 -14147.819,E2 -14147.819} C_VEL
LIN {X 0,Y 346.433,Z 353.298,A -85,B 0,C 180,E1 -14149.558,E2 -14149.558} C_VEL
LIN {X 0,Y 348.46,Z 342.103,A -85,B 0,C 180,E1 -14151.133,E2 -14151.133} C_VEL
LIN {X 0,Y 350.307,Z 331.017,A -85,B 0,C 180,E1 -14152.409,E2 -14152.409} C_VEL
LIN {X 0,Y 352.056,Z 318.983,A -85,B 0,C 180,E1 -14153.533,E2 -14153.533} C_VEL
LIN {X 0,Y 353.746,Z 305.68,A -85,B 0,C 180,E1 -14154.504,E2 -14154.504} C_VEL
LIN {X 0,Y 355.01,Z 293.372,A -85,B 0,C 180,E1 -14155.192,E2 -14155.192} C_VEL
LIN {X 0,Y 356.226,Z 278.564,A -85,B 0,C 180,E1 -14155.765,E2 -14155.765} C_VEL
LIN {X 0,Y 356.926,Z 261.102,A -85,B 0,C 180,E1 -14156.181,E2 -14156.181} C_VEL
LIN {X 0,Y 359.178,Z 180.723,A -85,B 0,C 180,E1 -14157.839,E2 -14157.839} C_VEL
LIN {X 0,Y 356.174,Z 163.854,A -85,B 0,C 180,E1 -14158.544,E2 -14158.544} C_VEL
LIN {X 0,Y 353.263,Z 150.923,A -85,B 0,C 180,E1 -14159.161,E2 -14159.161} C_VEL
LIN {X 0,Y 347.921,Z 139.495,A -85,B 0,C 180,E1 -14160.031,E2 -14160.031} C_VEL
LIN {X 0,Y 346.75,Z 136.683,A -85,B 0,C 180,E1 -14160.258,E2 -14160.258} C_VEL
LIN {X 0,Y 343.666,Z 124.162,A -85,B 0,C 180,E1 -14163.849,E2 -14163.849} C_VEL
LIN {X 0,Y 340.731,Z 113.661,A -85,B 0,C 180,E1 -14167.156,E2 -14167.156} C_VEL
LIN {X 0,Y 340.695,Z 113.665,A -85,B 0,C 180,E1 -14171.31,E2 -14171.31} C_VEL
LIN {X 0,Y 340.656,Z 113.677,A -85,B 0,C 180,E1 -14174.545,E2 -14174.545} C_VEL
LIN {X 0,Y 340.712,Z 113.652,A -85,B 0,C 180,E1 -14177.954,E2 -14177.954} C_VEL
LIN {X 0,Y 340.734,Z 113.666,A -85,B 0,C 180,E1 -14181.77,E2 -14181.77} C_VEL
LIN {X 0,Y 340.737,Z 113.661,A -85,B 0,C 180,E1 -14185.594,E2 -14185.594} C_VEL
LIN {X 0,Y 340.708,Z 113.664,A -85,B 0,C 180,E1 -14188.953,E2 -14188.953} C_VEL
LIN {X 0,Y 340.738,Z 113.66,A -85,B 0,C 180,E1 -14193.011,E2 -14193.011} C_VEL
LIN {X 0,Y 340.757,Z 113.655,A -85,B 0,C 180,E1 -14195.635,E2 -14195.635} C_VEL
LIN {X 0,Y 340.744,Z 113.656,A -85,B 0,C 180,E1 -14199.471,E2 -14199.471} C_VEL
LIN {X 0,Y 340.871,Z 113.649,A -85,B 0,C 180,E1 -14201.982,E2 -14201.982} C_VEL
LIN {X 0,Y 340.883,Z 113.647,A -85,B 0,C 180,E1 -14205.702,E2 -14205.702} C_VEL
LIN {X 0,Y 340.859,Z 113.649,A -85,B 0,C 180,E1 -14209.302,E2 -14209.302} C_VEL
LIN {X 0,Y 341.013,Z 113.624,A -85,B 0,C 180,E1 -14212.893,E2 -14212.893} C_VEL
LIN {X 0,Y 340.836,Z 113.652,A -85,B 0,C 180,E1 -14215.265,E2 -14215.265} C_VEL
LIN {X 0,Y 341.166,Z 113.605,A -85,B 0,C 180,E1 -14217.635,E2 -14217.635} C_VEL
LIN {X 0,Y 341.262,Z 113.598,A -85,B 0,C 180,E1 -14219.996,E2 -14219.996} C_VEL
LIN {X 0,Y 341.171,Z 113.61,A -85,B 0,C 180,E1 -14222.357,E2 -14222.357} C_VEL
LIN {X 0,Y 341.021,Z 113.63,A -85,B 0,C 180,E1 -14227.099,E2 -14227.099} C_VEL
LIN {X 0,Y 340.851,Z 113.65,A -85,B 0,C 180,E1 -14230.69,E2 -14230.69} C_VEL
LIN {X 0,Y 340.865,Z 113.65,A -85,B 0,C 180,E1 -14234.32,E2 -14234.32} C_VEL
LIN {X 0,Y 340.836,Z 113.653,A -85,B 0,C 180,E1 -14238.462,E2 -14238.462} C_VEL
LIN {X 0,Y 340.751,Z 113.665,A -85,B 0,C 180,E1 -14241.852,E2 -14241.852} C_VEL
LIN {X 0,Y 340.766,Z 113.658,A -85,B 0,C 180,E1 -14245.66,E2 -14245.66} C_VEL
LIN {X 0,Y 340.712,Z 113.665,A -85,B 0,C 180,E1 -14248.317,E2 -14248.317} C_VEL
LIN {X 0,Y 340.687,Z 113.662,A -85,B 0,C 180,E1 -14251.04,E2 -14251.04} C_VEL
LIN {X 0,Y 340.707,Z 113.664,A -85,B 0,C 180,E1 -14255.274,E2 -14255.274} C_VEL
LIN {X 0,Y 340.696,Z 113.663,A -85,B 0,C 180,E1 -14258.381,E2 -14258.381} C_VEL
LIN {X 0,Y 340.709,Z 113.824,A -85,B 0,C 180,E1 -14260.717,E2 -14260.717} C_VEL
LIN {X 0,Y 342.877,Z 121.853,A -85,B 0,C 180,E1 -14263.359,E2 -14263.359} C_VEL
LIN {X 0,Y 352.971,Z 141.322,A -85,B 0,C 180,E1 -14264.998,E2 -14264.998} C_VEL
LIN {X 0,Y 358.877,Z 154.365,A -85,B 0,C 180,E1 -14265.933,E2 -14265.933} C_VEL
LIN {X 0,Y 359.877,Z 157.458,A -85,B 0,C 180,E1 -14266.108,E2 -14266.108} C_VEL
LIN {X 0,Y 356.859,Z 257.796,A -85,B 0,C 180,E1 -14268.191,E2 -14268.191} C_VEL
LIN {X 0,Y 355.937,Z 272.383,A -85,B 0,C 180,E1 -14268.716,E2 -14268.716} C_VEL
LIN {X 0,Y 354.696,Z 286.191,A -85,B 0,C 180,E1 -14269.445,E2 -14269.445} C_VEL
LIN {X 0,Y 353.16,Z 300.098,A -85,B 0,C 180,E1 -14270.444,E2 -14270.444} C_VEL
LIN {X 0,Y 351.516,Z 311.791,A -85,B 0,C 180,E1 -14271.51,E2 -14271.51} C_VEL
LIN {X 0,Y 349.776,Z 322.801,A -85,B 0,C 180,E1 -14272.748,E2 -14272.748} C_VEL
LIN {X 0,Y 347.824,Z 334.102,A -85,B 0,C 180,E1 -14274.306,E2 -14274.306} C_VEL
LIN {X 0,Y 345.938,Z 344.259,A -85,B 0,C 180,E1 -14276.024,E2 -14276.024} C_VEL
LIN {X 0,Y 344.169,Z 353.437,A -85,B 0,C 180,E1 -14277.93,E2 -14277.93} C_VEL
LIN {X 0,Y 342.634,Z 361.193,A -85,B 0,C 180,E1 -14279.919,E2 -14279.919} C_VEL
LIN {X 0,Y 341.543,Z 367.006,A -85,B 0,C 180,E1 -14281.751,E2 -14281.751} C_VEL
LIN {X 0,Y 340.637,Z 371.911,A -85,B 0,C 180,E1 -14283.665,E2 -14283.665} C_VEL
LIN {X 0,Y 339.981,Z 375.779,A -85,B 0,C 180,E1 -14285.578,E2 -14285.578} C_VEL
LIN {X 0,Y 339.364,Z 379.46,A -85,B 0,C 180,E1 -14288.112,E2 -14288.112} C_VEL
LIN {X 0,Y 338.989,Z 381.588,A -85,B 0,C 180,E1 -14290.625,E2 -14290.625} C_VEL
LIN {X 0,Y 338.87,Z 382.229,A -85,B 0,C 180,E1 -14293.119,E2 -14293.119} C_VEL
LIN {X 0,Y 338.847,Z 381.429,A -85,B 0,C 180,E1 -14295.586,E2 -14295.586} C_VEL
LIN {X 0,Y 338.997,Z 379.224,A -85,B 0,C 180,E1 -14298.033,E2 -14298.033} C_VEL
LIN {X 0,Y 339.3,Z 375.588,A -85,B 0,C 180,E1 -14300.46,E2 -14300.46} C_VEL
LIN {X 0,Y 339.746,Z 370.437,A -85,B 0,C 180,E1 -14302.869,E2 -14302.869} C_VEL
LIN {X 0,Y 340.222,Z 365.448,A -85,B 0,C 180,E1 -14304.665,E2 -14304.665} C_VEL
LIN {X 0,Y 341.054,Z 358.294,A -85,B 0,C 180,E1 -14306.75,E2 -14306.75} C_VEL
LIN {X 0,Y 342.005,Z 350.811,A -85,B 0,C 180,E1 -14308.526,E2 -14308.526} C_VEL
LIN {X 0,Y 343.195,Z 341.824,A -85,B 0,C 180,E1 -14310.292,E2 -14310.292} C_VEL
LIN {X 0,Y 344.549,Z 331.162,A -85,B 0,C 180,E1 -14312.014,E2 -14312.014} C_VEL
LIN {X 0,Y 345.864,Z 319.959,A -85,B 0,C 180,E1 -14313.493,E2 -14313.493} C_VEL
LIN {X 0,Y 347.215,Z 307.861,A -85,B 0,C 180,E1 -14314.788,E2 -14314.788} C_VEL
LIN {X 0,Y 348.484,Z 294.323,A -85,B 0,C 180,E1 -14315.931,E2 -14315.931} C_VEL
LIN {X 0,Y 349.495,Z 281.217,A -85,B 0,C 180,E1 -14316.783,E2 -14316.783} C_VEL
LIN {X 0,Y 350.303,Z 267.08,A -85,B 0,C 180,E1 -14317.455,E2 -14317.455} C_VEL
LIN {X 0,Y 350.756,Z 253.666,A -85,B 0,C 180,E1 -14317.88,E2 -14317.88} C_VEL
LIN {X 0,Y 353.149,Z 153.386,A -85,B 0,C 180,E1 -14319.921,E2 -14319.921} C_VEL
LIN {X 0,Y 351.155,Z 144.193,A -85,B 0,C 180,E1 -14320.255,E2 -14320.255} C_VEL
LIN {X 0,Y 342.624,Z 121.633,A -85,B 0,C 180,E1 -14321.351,E2 -14321.351} C_VEL
LIN {X 0,Y 341.576,Z 120.497,A -85,B 0,C 180,E1 -14321.54,E2 -14321.54} C_VEL
LIN {X 0,Y 336.706,Z 117.569,A -85,B 0,C 180,E1 -14322.746,E2 -14322.746} C_VEL
LIN {X 0,Y 334.278,Z 115.152,A -85,B 0,C 180,E1 -14323.775,E2 -14323.775} C_VEL
LIN {X 0,Y 333.788,Z 114.535,A -85,B 0,C 180,E1 -14324.407,E2 -14324.407} C_VEL
LIN {X 0,Y 333.768,Z 114.533,A -85,B 0,C 180,E1 -14328.659,E2 -14328.659} C_VEL
LIN {X 0,Y 333.698,Z 114.541,A -85,B 0,C 180,E1 -14332.276,E2 -14332.276} C_VEL
LIN {X 0,Y 333.695,Z 114.544,A -85,B 0,C 180,E1 -14335.106,E2 -14335.106} C_VEL
LIN {X 0,Y 333.687,Z 114.542,A -85,B 0,C 180,E1 -14337.811,E2 -14337.811} C_VEL
LIN {X 0,Y 333.666,Z 114.544,A -85,B 0,C 180,E1 -14340.363,E2 -14340.363} C_VEL
LIN {X 0,Y 333.655,Z 114.548,A -85,B 0,C 180,E1 -14344.659,E2 -14344.659} C_VEL
LIN {X 0,Y 333.684,Z 114.542,A -85,B 0,C 180,E1 -14347.644,E2 -14347.644} C_VEL
LIN {X 0,Y 333.72,Z 114.542,A -85,B 0,C 180,E1 -14350.754,E2 -14350.754} C_VEL
LIN {X 0,Y 333.709,Z 114.537,A -85,B 0,C 180,E1 -14354.279,E2 -14354.279} C_VEL
LIN {X 0,Y 333.677,Z 114.542,A -85,B 0,C 180,E1 -14357.631,E2 -14357.631} C_VEL
LIN {X 0,Y 333.655,Z 114.542,A -85,B 0,C 180,E1 -14361.198,E2 -14361.198} C_VEL
LIN {X 0,Y 333.659,Z 114.545,A -85,B 0,C 180,E1 -14365.229,E2 -14365.229} C_VEL
LIN {X 0,Y 333.62,Z 114.554,A -85,B 0,C 180,E1 -14368.227,E2 -14368.227} C_VEL
LIN {X 0,Y 333.688,Z 114.537,A -85,B 0,C 180,E1 -14371.031,E2 -14371.031} C_VEL
LIN {X 0,Y 333.716,Z 114.537,A -85,B 0,C 180,E1 -14373.757,E2 -14373.757} C_VEL
LIN {X 0,Y 333.697,Z 114.543,A -85,B 0,C 180,E1 -14376.417,E2 -14376.417} C_VEL
LIN {X 0,Y 333.739,Z 114.537,A -85,B 0,C 180,E1 -14380.315,E2 -14380.315} C_VEL
LIN {X 0,Y 333.761,Z 114.534,A -85,B 0,C 180,E1 -14384.118,E2 -14384.118} C_VEL
LIN {X 0,Y 333.78,Z 114.534,A -85,B 0,C 180,E1 -14387.849,E2 -14387.849} C_VEL
LIN {X 0,Y 333.983,Z 114.508,A -85,B 0,C 180,E1 -14391.534,E2 -14391.534} C_VEL
LIN {X 0,Y 334.009,Z 114.499,A -85,B 0,C 180,E1 -14393.965,E2 -14393.965} C_VEL
LIN {X 0,Y 334.121,Z 114.491,A -85,B 0,C 180,E1 -14397.593,E2 -14397.593} C_VEL
LIN {X 0,Y 334.257,Z 114.471,A -85,B 0,C 180,E1 -14400.004,E2 -14400.004} C_VEL
LIN {X 0,Y 334.098,Z 114.489,A -85,B 0,C 180,E1 -14402.415,E2 -14402.415} C_VEL
LIN {X 0,Y 334.017,Z 114.504,A -85,B 0,C 180,E1 -14407.256,E2 -14407.256} C_VEL
LIN {X 0,Y 333.827,Z 114.529,A -85,B 0,C 180,E1 -14410.926,E2 -14410.926} C_VEL
LIN {X 0,Y 333.802,Z 114.53,A -85,B 0,C 180,E1 -14414.638,E2 -14414.638} C_VEL
LIN {X 0,Y 333.792,Z 114.533,A -85,B 0,C 180,E1 -14418.659,E2 -14418.659} C_VEL
LIN {X 0,Y 333.689,Z 114.543,A -85,B 0,C 180,E1 -14422.282,E2 -14422.282} C_VEL
LIN {X 0,Y 333.733,Z 114.539,A -85,B 0,C 180,E1 -14426.25,E2 -14426.25} C_VEL
LIN {X 0,Y 333.709,Z 114.54,A -85,B 0,C 180,E1 -14428.976,E2 -14428.976} C_VEL
LIN {X 0,Y 333.642,Z 114.55,A -85,B 0,C 180,E1 -14432.59,E2 -14432.59} C_VEL
LIN {X 0,Y 333.676,Z 114.548,A -85,B 0,C 180,E1 -14436.142,E2 -14436.142} C_VEL
LIN {X 0,Y 333.647,Z 114.546,A -85,B 0,C 180,E1 -14439.196,E2 -14439.196} C_VEL
LIN {X 0,Y 333.634,Z 114.55,A -85,B 0,C 180,E1 -14442.503,E2 -14442.503} C_VEL
LIN {X 0,Y 333.598,Z 114.558,A -85,B 0,C 180,E1 -14445.958,E2 -14445.958} C_VEL
LIN {X 0,Y 333.65,Z 114.547,A -85,B 0,C 180,E1 -14449.319,E2 -14449.319} C_VEL
LIN {X 0,Y 333.668,Z 114.547,A -85,B 0,C 180,E1 -14453.171,E2 -14453.171} C_VEL
LIN {X 0,Y 333.69,Z 114.694,A -85,B 0,C 180,E1 -14456.574,E2 -14456.574} C_VEL
LIN {X 0,Y 336.616,Z 127.605,A -85,B 0,C 180,E1 -14459.931,E2 -14459.931} C_VEL
LIN {X 0,Y 338.683,Z 137.61,A -85,B 0,C 180,E1 -14462.368,E2 -14462.368} C_VEL
LIN {X 0,Y 340.353,Z 143.291,A -85,B 0,C 180,E1 -14462.617,E2 -14462.617} C_VEL
LIN {X 0,Y 346.12,Z 179.434,A -85,B 0,C 180,E1 -14463.824,E2 -14463.824} C_VEL
LIN {X 0,Y 343.921,Z 275.246,A -85,B 0,C 180,E1 -14465.839,E2 -14465.839} C_VEL
LIN {X 0,Y 343.14,Z 289.214,A -85,B 0,C 180,E1 -14466.342,E2 -14466.342} C_VEL
LIN {X 0,Y 342.041,Z 303.483,A -85,B 0,C 180,E1 -14467.103,E2 -14467.103} C_VEL
LIN {X 0,Y 340.985,Z 314.907,A -85,B 0,C 180,E1 -14467.907,E2 -14467.907} C_VEL
LIN {X 0,Y 339.67,Z 327.053,A -85,B 0,C 180,E1 -14468.985,E2 -14468.985} C_VEL
LIN {X 0,Y 338.397,Z 337.515,A -85,B 0,C 180,E1 -14470.12,E2 -14470.12} C_VEL
LIN {X 0,Y 336.958,Z 348.782,A -85,B 0,C 180,E1 -14471.613,E2 -14471.613} C_VEL
LIN {X 0,Y 335.626,Z 359.025,A -85,B 0,C 180,E1 -14473.268,E2 -14473.268} C_VEL
LIN {X 0,Y 334.468,Z 368.586,A -85,B 0,C 180,E1 -14475.152,E2 -14475.152} C_VEL
LIN {X 0,Y 333.574,Z 375.991,A -85,B 0,C 180,E1 -14476.911,E2 -14476.911} C_VEL
LIN {X 0,Y 332.747,Z 383.318,A -85,B 0,C 180,E1 -14479.044,E2 -14479.044} C_VEL
LIN {X 0,Y 332.371,Z 388.444,A -85,B 0,C 180,E1 -14480.877,E2 -14480.877} C_VEL
LIN {X 0,Y 332.039,Z 393.698,A -85,B 0,C 180,E1 -14483.317,E2 -14483.317} C_VEL
LIN {X 0,Y 331.937,Z 396.638,A -85,B 0,C 180,E1 -14485.144,E2 -14485.144} C_VEL
LIN {X 0,Y 331.978,Z 398.14,A -85,B 0,C 180,E1 -14486.36,E2 -14486.36} C_VEL
LIN {X 0,Y 331.928,Z 400.072,A -85,B 0,C 180,E1 -14488.789,E2 -14488.789} C_VEL
LIN {X 0,Y 331.974,Z 400.526,A -85,B 0,C 180,E1 -14490.002,E2 -14490.002} C_VEL
LIN {X 0,Y 331.913,Z 400.421,A -85,B 0,C 180,E1 -14492.429,E2 -14492.429} C_VEL
LIN {X 0,Y 331.953,Z 398.987,A -85,B 0,C 180,E1 -14494.86,E2 -14494.86} C_VEL
LIN {X 0,Y 332.181,Z 396.203,A -85,B 0,C 180,E1 -14497.295,E2 -14497.295} C_VEL
LIN {X 0,Y 332.673,Z 391.999,A -85,B 0,C 180,E1 -14499.732,E2 -14499.732} C_VEL
LIN {X 0,Y 333.512,Z 386.261,A -85,B 0,C 180,E1 -14502.167,E2 -14502.167} C_VEL
LIN {X 0,Y 334.691,Z 379.826,A -85,B 0,C 180,E1 -14504.286,E2 -14504.286} C_VEL
LIN {X 0,Y 336.12,Z 371.869,A -85,B 0,C 180,E1 -14506.398,E2 -14506.398} C_VEL
LIN {X 0,Y 337.761,Z 363.573,A -85,B 0,C 180,E1 -14508.188,E2 -14508.188} C_VEL
LIN {X 0,Y 339.765,Z 353.615,A -85,B 0,C 180,E1 -14509.958,E2 -14509.958} C_VEL
LIN {X 0,Y 341.878,Z 342.564,A -85,B 0,C 180,E1 -14511.561,E2 -14511.561} C_VEL
LIN {X 0,Y 343.989,Z 330.291,A -85,B 0,C 180,E1 -14512.995,E2 -14512.995} C_VEL
LIN {X 0,Y 345.874,Z 318.067,A -85,B 0,C 180,E1 -14514.139,E2 -14514.139} C_VEL
LIN {X 0,Y 347.587,Z 304.593,A -85,B 0,C 180,E1 -14515.127,E2 -14515.127} C_VEL
LIN {X 0,Y 349.108,Z 290.482,A -85,B 0,C 180,E1 -14515.889,E2 -14515.889} C_VEL
LIN {X 0,Y 350.267,Z 276.6,A -85,B 0,C 180,E1 -14516.397,E2 -14516.397} C_VEL
LIN {X 0,Y 351.157,Z 249.646,A -85,B 0,C 180,E1 -14517.006,E2 -14517.006} C_VEL
LIN {X 0,Y 353.135,Z 181.207,A -85,B 0,C 180,E1 -14518.444,E2 -14518.444} C_VEL
LIN {X 0,Y 349.403,Z 161.129,A -85,B 0,C 180,E1 -14519.329,E2 -14519.329} C_VEL
LIN {X 0,Y 347.509,Z 153.557,A -85,B 0,C 180,E1 -14519.726,E2 -14519.726} C_VEL
LIN {X 0,Y 341.255,Z 140.242,A -85,B 0,C 180,E1 -14520.786,E2 -14520.786} C_VEL
LIN {X 0,Y 339.493,Z 136.401,A -85,B 0,C 180,E1 -14521.125,E2 -14521.125} C_VEL
LIN {X 0,Y 336.531,Z 124.633,A -85,B 0,C 180,E1 -14524.637,E2 -14524.637} C_VEL
LIN {X 0,Y 333.706,Z 114.536,A -85,B 0,C 180,E1 -14527.932,E2 -14527.932} C_VEL
LIN {X 0,Y 333.658,Z 114.537,A -85,B 0,C 180,E1 -14530.768,E2 -14530.768} C_VEL
LIN {X 0,Y 333.609,Z 114.557,A -85,B 0,C 180,E1 -14534.249,E2 -14534.249} C_VEL
LIN {X 0,Y 333.656,Z 114.535,A -85,B 0,C 180,E1 -14537.617,E2 -14537.617} C_VEL
LIN {X 0,Y 333.655,Z 114.549,A -85,B 0,C 180,E1 -14541.204,E2 -14541.204} C_VEL
LIN {X 0,Y 333.689,Z 114.545,A -85,B 0,C 180,E1 -14543.859,E2 -14543.859} C_VEL
LIN {X 0,Y 333.659,Z 114.55,A -85,B 0,C 180,E1 -14547.412,E2 -14547.412} C_VEL
LIN {X 0,Y 333.669,Z 114.548,A -85,B 0,C 180,E1 -14551.021,E2 -14551.021} C_VEL
LIN {X 0,Y 333.714,Z 114.537,A -85,B 0,C 180,E1 -14555.086,E2 -14555.086} C_VEL
LIN {X 0,Y 333.685,Z 114.539,A -85,B 0,C 180,E1 -14559.016,E2 -14559.016} C_VEL
LIN {X 0,Y 333.807,Z 114.529,A -85,B 0,C 180,E1 -14561.587,E2 -14561.587} C_VEL
LIN {X 0,Y 333.822,Z 114.527,A -85,B 0,C 180,E1 -14565.574,E2 -14565.574} C_VEL
LIN {X 0,Y 333.829,Z 114.522,A -85,B 0,C 180,E1 -14569.074,E2 -14569.074} C_VEL
LIN {X 0,Y 333.968,Z 114.501,A -85,B 0,C 180,E1 -14572.743,E2 -14572.743} C_VEL
LIN {X 0,Y 333.801,Z 114.529,A -85,B 0,C 180,E1 -14575.165,E2 -14575.165} C_VEL
LIN {X 0,Y 334.102,Z 114.484,A -85,B 0,C 180,E1 -14577.585,E2 -14577.585} C_VEL
LIN {X 0,Y 334.214,Z 114.476,A -85,B 0,C 180,E1 -14579.996,E2 -14579.996} C_VEL
LIN {X 0,Y 334.108,Z 114.49,A -85,B 0,C 180,E1 -14582.407,E2 -14582.407} C_VEL
LIN {X 0,Y 333.974,Z 114.502,A -85,B 0,C 180,E1 -14586.506,E2 -14586.506} C_VEL
LIN {X 0,Y 333.824,Z 114.52,A -85,B 0,C 180,E1 -14589.692,E2 -14589.692} C_VEL
LIN {X 0,Y 333.799,Z 114.523,A -85,B 0,C 180,E1 -14593.387,E2 -14593.387} C_VEL
LIN {X 0,Y 333.746,Z 114.53,A -85,B 0,C 180,E1 -14597.141,E2 -14597.141} C_VEL
LIN {X 0,Y 333.735,Z 114.533,A -85,B 0,C 180,E1 -14599.686,E2 -14599.686} C_VEL
LIN {X 0,Y 333.689,Z 114.543,A -85,B 0,C 180,E1 -14602.273,E2 -14602.273} C_VEL
LIN {X 0,Y 333.724,Z 114.534,A -85,B 0,C 180,E1 -14606.242,E2 -14606.242} C_VEL
LIN {X 0,Y 333.675,Z 114.531,A -85,B 0,C 180,E1 -14608.97,E2 -14608.97} C_VEL
LIN {X 0,Y 333.627,Z 114.544,A -85,B 0,C 180,E1 -14613.203,E2 -14613.203} C_VEL
LIN {X 0,Y 333.664,Z 114.551,A -85,B 0,C 180,E1 -14616.134,E2 -14616.134} C_VEL
LIN {X 0,Y 333.684,Z 114.712,A -85,B 0,C 180,E1 -14619.963,E2 -14619.963} C_VEL
LIN {X 0,Y 335.664,Z 122.093,A -85,B 0,C 180,E1 -14622.479,E2 -14622.479} C_VEL
LIN {X 0,Y 344.288,Z 138.22,A -85,B 0,C 180,E1 -14623.944,E2 -14623.944} C_VEL
LIN {X 0,Y 351.735,Z 153.695,A -85,B 0,C 180,E1 -14625.165,E2 -14625.165} C_VEL
LIN {X 0,Y 353.902,Z 158.898,A -85,B 0,C 180,E1 -14625.522,E2 -14625.522} C_VEL
LIN {X 0,Y 350.769,Z 257.524,A -85,B 0,C 180,E1 -14627.594,E2 -14627.594} C_VEL
LIN {X 0,Y 349.847,Z 271.857,A -85,B 0,C 180,E1 -14628.105,E2 -14628.105} C_VEL
LIN {X 0,Y 348.523,Z 286.071,A -85,B 0,C 180,E1 -14628.859,E2 -14628.859} C_VEL
LIN {X 0,Y 347.066,Z 298.803,A -85,B 0,C 180,E1 -14629.771,E2 -14629.771} C_VEL
LIN {X 0,Y 345.306,Z 311.026,A -85,B 0,C 180,E1 -14630.879,E2 -14630.879} C_VEL
LIN {X 0,Y 343.269,Z 323.422,A -85,B 0,C 180,E1 -14632.289,E2 -14632.289} C_VEL
LIN {X 0,Y 341.22,Z 334.641,A -85,B 0,C 180,E1 -14633.871,E2 -14633.871} C_VEL
LIN {X 0,Y 339.249,Z 344.788,A -85,B 0,C 180,E1 -14635.629,E2 -14635.629} C_VEL
LIN {X 0,Y 337.39,Z 353.853,A -85,B 0,C 180,E1 -14637.56,E2 -14637.56} C_VEL
LIN {X 0,Y 335.932,Z 360.935,A -85,B 0,C 180,E1 -14639.402,E2 -14639.402} C_VEL
LIN {X 0,Y 334.547,Z 367.796,A -85,B 0,C 180,E1 -14641.617,E2 -14641.617} C_VEL
LIN {X 0,Y 333.53,Z 372.966,A -85,B 0,C 180,E1 -14643.735,E2 -14643.735} C_VEL
LIN {X 0,Y 333.027,Z 375.69,A -85,B 0,C 180,E1 -14645.141,E2 -14645.141} C_VEL
LIN {X 0,Y 332.365,Z 379.34,A -85,B 0,C 180,E1 -14647.626,E2 -14647.626} C_VEL
LIN {X 0,Y 331.93,Z 381.613,A -85,B 0,C 180,E1 -14650.196,E2 -14650.196} C_VEL
LIN {X 0,Y 331.788,Z 382.417,A -85,B 0,C 180,E1 -14652.748,E2 -14652.748} C_VEL
LIN {X 0,Y 331.743,Z 381.796,A -85,B 0,C 180,E1 -14655.271,E2 -14655.271} C_VEL
LIN {X 0,Y 331.893,Z 379.736,A -85,B 0,C 180,E1 -14657.773,E2 -14657.773} C_VEL
LIN {X 0,Y 332.183,Z 376.242,A -85,B 0,C 180,E1 -14660.254,E2 -14660.254} C_VEL
LIN {X 0,Y 332.631,Z 371.24,A -85,B 0,C 180,E1 -14662.715,E2 -14662.715} C_VEL
LIN {X 0,Y 333.102,Z 366.412,A -85,B 0,C 180,E1 -14664.55,E2 -14664.55} C_VEL
LIN {X 0,Y 333.932,Z 359.43,A -85,B 0,C 180,E1 -14666.68,E2 -14666.68} C_VEL
LIN {X 0,Y 335.059,Z 350.784,A -85,B 0,C 180,E1 -14668.796,E2 -14668.796} C_VEL
LIN {X 0,Y 336.313,Z 341.745,A -85,B 0,C 180,E1 -14670.597,E2 -14670.597} C_VEL
LIN {X 0,Y 337.552,Z 332.183,A -85,B 0,C 180,E1 -14672.177,E2 -14672.177} C_VEL
LIN {X 0,Y 338.92,Z 320.921,A -85,B 0,C 180,E1 -14673.714,E2 -14673.714} C_VEL
LIN {X 0,Y 340.314,Z 308.992,A -85,B 0,C 180,E1 -14675.034,E2 -14675.034} C_VEL
LIN {X 0,Y 341.647,Z 295.78,A -85,B 0,C 180,E1 -14676.198,E2 -14676.198} C_VEL
LIN {X 0,Y 342.666,Z 283.077,A -85,B 0,C 180,E1 -14677.067,E2 -14677.067} C_VEL
LIN {X 0,Y 343.54,Z 268.713,A -85,B 0,C 180,E1 -14677.788,E2 -14677.788} C_VEL
LIN {X 0,Y 344.069,Z 254.716,A -85,B 0,C 180,E1 -14678.256,E2 -14678.256} C_VEL
LIN {X 0,Y 346.473,Z 153.855,A -85,B 0,C 180,E1 -14680.358,E2 -14680.358} C_VEL
LIN {X 0,Y 344.786,Z 146.377,A -85,B 0,C 180,E1 -14680.641,E2 -14680.641} C_VEL
LIN {X 0,Y 336.253,Z 123.828,A -85,B 0,C 180,E1 -14681.765,E2 -14681.765} C_VEL
LIN {X 0,Y 335.187,Z 121.031,A -85,B 0,C 180,E1 -14681.912,E2 -14681.912} C_VEL
LIN {X 0,Y 333.85,Z 114.53,A -85,B 0,C 180,E1 -14683.773,E2 -14683.773} C_VEL
LIN {X 0,Y 333.788,Z 114.535,A -85,B 0,C 180,E1 -14684.407,E2 -14684.407} C_VEL
LIN {X 0,Y 333.063,Z 114.627,A -85,B 0,C 180,E1 -14685.413,E2 -14685.413} C_VEL
LIN {X 0,Y 330.193,Z 114.981,A -85,B 0,C 180,E1 -14687.05,E2 -14687.05} C_VEL
LIN {X 0,Y 327.789,Z 115.278,A -85,B 0,C 180,E1 -14688.377,E2 -14688.377} C_VEL
LIN {X 0,Y 326.75,Z 115.412,A -85,B 0,C 180,E1 -14689.403,E2 -14689.403} C_VEL
LIN {X 0,Y 326.66,Z 115.417,A -85,B 0,C 180,E1 -14689.751,E2 -14689.751} C_VEL
LIN {X 0,Y 326.653,Z 115.419,A -85,B 0,C 180,E1 -14692.783,E2 -14692.783} C_VEL
LIN {X 0,Y 326.652,Z 115.42,A -85,B 0,C 180,E1 -14696.858,E2 -14696.858} C_VEL
LIN {X 0,Y 326.608,Z 115.424,A -85,B 0,C 180,E1 -14700.613,E2 -14700.613} C_VEL
LIN {X 0,Y 326.585,Z 115.426,A -85,B 0,C 180,E1 -14704.02,E2 -14704.02} C_VEL
LIN {X 0,Y 326.652,Z 115.421,A -85,B 0,C 180,E1 -14707.253,E2 -14707.253} C_VEL
LIN {X 0,Y 326.644,Z 115.421,A -85,B 0,C 180,E1 -14711.153,E2 -14711.153} C_VEL
LIN {X 0,Y 326.65,Z 115.418,A -85,B 0,C 180,E1 -14715.233,E2 -14715.233} C_VEL
LIN {X 0,Y 326.604,Z 115.426,A -85,B 0,C 180,E1 -14718.86,E2 -14718.86} C_VEL
LIN {X 0,Y 326.62,Z 115.417,A -85,B 0,C 180,E1 -14721.398,E2 -14721.398} C_VEL
LIN {X 0,Y 326.593,Z 115.427,A -85,B 0,C 180,E1 -14724.854,E2 -14724.854} C_VEL
LIN {X 0,Y 326.59,Z 115.425,A -85,B 0,C 180,E1 -14727.46,E2 -14727.46} C_VEL
LIN {X 0,Y 326.638,Z 115.418,A -85,B 0,C 180,E1 -14730.345,E2 -14730.345} C_VEL
LIN {X 0,Y 326.671,Z 115.417,A -85,B 0,C 180,E1 -14734.52,E2 -14734.52} C_VEL
LIN {X 0,Y 326.655,Z 115.418,A -85,B 0,C 180,E1 -14738.551,E2 -14738.551} C_VEL
LIN {X 0,Y 326.725,Z 115.409,A -85,B 0,C 180,E1 -14741.181,E2 -14741.181} C_VEL
LIN {X 0,Y 326.746,Z 115.407,A -85,B 0,C 180,E1 -14745.437,E2 -14745.437} C_VEL
LIN {X 0,Y 326.758,Z 115.405,A -85,B 0,C 180,E1 -14748.843,E2 -14748.843} C_VEL
LIN {X 0,Y 326.966,Z 115.374,A -85,B 0,C 180,E1 -14752.594,E2 -14752.594} C_VEL
LIN {X 0,Y 326.77,Z 115.4,A -85,B 0,C 180,E1 -14755.069,E2 -14755.069} C_VEL
LIN {X 0,Y 327.058,Z 115.371,A -85,B 0,C 180,E1 -14757.541,E2 -14757.541} C_VEL
LIN {X 0,Y 327.208,Z 115.349,A -85,B 0,C 180,E1 -14760.004,E2 -14760.004} C_VEL
LIN {X 0,Y 327.038,Z 115.368,A -85,B 0,C 180,E1 -14762.467,E2 -14762.467} C_VEL
LIN {X 0,Y 326.988,Z 115.373,A -85,B 0,C 180,E1 -14766.173,E2 -14766.173} C_VEL
LIN {X 0,Y 326.907,Z 115.387,A -85,B 0,C 180,E1 -14768.659,E2 -14768.659} C_VEL
LIN {X 0,Y 326.728,Z 115.409,A -85,B 0,C 180,E1 -14772.425,E2 -14772.425} C_VEL
LIN {X 0,Y 326.748,Z 115.411,A -85,B 0,C 180,E1 -14774.961,E2 -14774.961} C_VEL
LIN {X 0,Y 326.729,Z 115.413,A -85,B 0,C 180,E1 -14778.842,E2 -14778.842} C_VEL
LIN {X 0,Y 326.617,Z 115.426,A -85,B 0,C 180,E1 -14782.791,E2 -14782.791} C_VEL
LIN {X 0,Y 326.688,Z 115.413,A -85,B 0,C 180,E1 -14785.487,E2 -14785.487} C_VEL
LIN {X 0,Y 326.659,Z 115.417,A -85,B 0,C 180,E1 -14789.663,E2 -14789.663} C_VEL
LIN {X 0,Y 326.606,Z 115.426,A -85,B 0,C 180,E1 -14794.023,E2 -14794.023} C_VEL
LIN {X 0,Y 326.627,Z 115.421,A -85,B 0,C 180,E1 -14797.242,E2 -14797.242} C_VEL
LIN {X 0,Y 326.579,Z 115.426,A -85,B 0,C 180,E1 -14801.135,E2 -14801.135} C_VEL
LIN {X 0,Y 326.529,Z 115.434,A -85,B 0,C 180,E1 -14804.746,E2 -14804.746} C_VEL
LIN {X 0,Y 326.579,Z 115.429,A -85,B 0,C 180,E1 -14808.157,E2 -14808.157} C_VEL
LIN {X 0,Y 326.626,Z 115.424,A -85,B 0,C 180,E1 -14811.394,E2 -14811.394} C_VEL
LIN {X 0,Y 326.623,Z 115.425,A -85,B 0,C 180,E1 -14814.855,E2 -14814.855} C_VEL
LIN {X 0,Y 326.639,Z 115.449,A -85,B 0,C 180,E1 -14816.131,E2 -14816.131} C_VEL
LIN {X 0,Y 329.578,Z 128.365,A -85,B 0,C 180,E1 -14819.575,E2 -14819.575} C_VEL
LIN {X 0,Y 331.396,Z 137.118,A -85,B 0,C 180,E1 -14821.811,E2 -14821.811} C_VEL
LIN {X 0,Y 333.942,Z 145.027,A -85,B 0,C 180,E1 -14822.194,E2 -14822.194} C_VEL
LIN {X 0,Y 339.534,Z 181.007,A -85,B 0,C 180,E1 -14823.416,E2 -14823.416} C_VEL
LIN {X 0,Y 337.271,Z 274.568,A -85,B 0,C 180,E1 -14825.413,E2 -14825.413} C_VEL
LIN {X 0,Y 336.492,Z 288.742,A -85,B 0,C 180,E1 -14825.927,E2 -14825.927} C_VEL
LIN {X 0,Y 335.329,Z 303.076,A -85,B 0,C 180,E1 -14826.699,E2 -14826.699} C_VEL
LIN {X 0,Y 334.163,Z 315.442,A -85,B 0,C 180,E1 -14827.594,E2 -14827.594} C_VEL
LIN {X 0,Y 332.625,Z 328.736,A -85,B 0,C 180,E1 -14828.826,E2 -14828.826} C_VEL
LIN {X 0,Y 331.238,Z 340.2,A -85,B 0,C 180,E1 -14830.157,E2 -14830.157} C_VEL
LIN {X 0,Y 329.739,Z 350.97,A -85,B 0,C 180,E1 -14831.679,E2 -14831.679} C_VEL
LIN {X 0,Y 328.317,Z 361.646,A -85,B 0,C 180,E1 -14833.525,E2 -14833.525} C_VEL
LIN {X 0,Y 327.268,Z 369.915,A -85,B 0,C 180,E1 -14835.265,E2 -14835.265} C_VEL
LIN {X 0,Y 326.386,Z 377.735,A -85,B 0,C 180,E1 -14837.251,E2 -14837.251} C_VEL
LIN {X 0,Y 325.554,Z 384.695,A -85,B 0,C 180,E1 -14839.428,E2 -14839.428} C_VEL
LIN {X 0,Y 325.201,Z 389.488,A -85,B 0,C 180,E1 -14841.301,E2 -14841.301} C_VEL
LIN {X 0,Y 324.902,Z 394.427,A -85,B 0,C 180,E1 -14843.793,E2 -14843.793} C_VEL
LIN {X 0,Y 324.881,Z 397.842,A -85,B 0,C 180,E1 -14846.281,E2 -14846.281} C_VEL
LIN {X 0,Y 324.836,Z 399.831,A -85,B 0,C 180,E1 -14848.762,E2 -14848.762} C_VEL
LIN {X 0,Y 324.879,Z 400.312,A -85,B 0,C 180,E1 -14850.002,E2 -14850.002} C_VEL
LIN {X 0,Y 324.832,Z 400.258,A -85,B 0,C 180,E1 -14852.482,E2 -14852.482} C_VEL
LIN {X 0,Y 324.869,Z 398.871,A -85,B 0,C 180,E1 -14854.966,E2 -14854.966} C_VEL
LIN {X 0,Y 325.112,Z 396.136,A -85,B 0,C 180,E1 -14857.454,E2 -14857.454} C_VEL
LIN {X 0,Y 325.622,Z 391.982,A -85,B 0,C 180,E1 -14859.945,E2 -14859.945} C_VEL
LIN {X 0,Y 326.563,Z 386.297,A -85,B 0,C 180,E1 -14862.43,E2 -14862.43} C_VEL
LIN {X 0,Y 327.755,Z 379.92,A -85,B 0,C 180,E1 -14864.595,E2 -14864.595} C_VEL
LIN {X 0,Y 329.277,Z 372.028,A -85,B 0,C 180,E1 -14866.748,E2 -14866.748} C_VEL
LIN {X 0,Y 331.025,Z 363.81,A -85,B 0,C 180,E1 -14868.572,E2 -14868.572} C_VEL
LIN {X 0,Y 333.117,Z 353.95,A -85,B 0,C 180,E1 -14870.374,E2 -14870.374} C_VEL
LIN {X 0,Y 335.311,Z 343.025,A -85,B 0,C 180,E1 -14872.005,E2 -14872.005} C_VEL
LIN {X 0,Y 337.479,Z 331.17,A -85,B 0,C 180,E1 -14873.441,E2 -14873.441} C_VEL
LIN {X 0,Y 339.469,Z 318.959,A -85,B 0,C 180,E1 -14874.625,E2 -14874.625} C_VEL
LIN {X 0,Y 341.35,Z 304.678,A -85,B 0,C 180,E1 -14875.701,E2 -14875.701} C_VEL
LIN {X 0,Y 342.957,Z 290.656,A -85,B 0,C 180,E1 -14876.47,E2 -14876.47} C_VEL
LIN {X 0,Y 344.14,Z 276.963,A -85,B 0,C 180,E1 -14876.986,E2 -14876.986} C_VEL
LIN {X 0,Y 344.922,Z 255.487,A -85,B 0,C 180,E1 -14877.494,E2 -14877.494} C_VEL
LIN {X 0,Y 347.142,Z 182.229,A -85,B 0,C 180,E1 -14879.057,E2 -14879.057} C_VEL
LIN {X 0,Y 343.069,Z 160.567,A -85,B 0,C 180,E1 -14880.054,E2 -14880.054} C_VEL
LIN {X 0,Y 341.89,Z 156.297,A -85,B 0,C 180,E1 -14880.299,E2 -14880.299} C_VEL
LIN {X 0,Y 335.903,Z 143.699,A -85,B 0,C 180,E1 -14881.344,E2 -14881.344} C_VEL
LIN {X 0,Y 332.211,Z 136.138,A -85,B 0,C 180,E1 -14882.041,E2 -14882.041} C_VEL
LIN {X 0,Y 329.695,Z 126.112,A -85,B 0,C 180,E1 -14885.14,E2 -14885.14} C_VEL
LIN {X 0,Y 326.636,Z 115.425,A -85,B 0,C 180,E1 -14888.761,E2 -14888.761} C_VEL
LIN {X 0,Y 326.591,Z 115.427,A -85,B 0,C 180,E1 -14892.971,E2 -14892.971} C_VEL
LIN {X 0,Y 326.59,Z 115.425,A -85,B 0,C 180,E1 -14897.028,E2 -14897.028} C_VEL
LIN {X 0,Y 326.614,Z 115.424,A -85,B 0,C 180,E1 -14900.775,E2 -14900.775} C_VEL
LIN {X 0,Y 326.626,Z 115.424,A -85,B 0,C 180,E1 -14904.479,E2 -14904.479} C_VEL
LIN {X 0,Y 326.623,Z 115.426,A -85,B 0,C 180,E1 -14907.454,E2 -14907.454} C_VEL
LIN {X 0,Y 326.631,Z 115.423,A -85,B 0,C 180,E1 -14910.335,E2 -14910.335} C_VEL
LIN {X 0,Y 326.658,Z 115.421,A -85,B 0,C 180,E1 -14914.642,E2 -14914.642} C_VEL
LIN {X 0,Y 326.632,Z 115.424,A -85,B 0,C 180,E1 -14918.541,E2 -14918.541} C_VEL
LIN {X 0,Y 326.759,Z 115.406,A -85,B 0,C 180,E1 -14921.175,E2 -14921.175} C_VEL
LIN {X 0,Y 326.777,Z 115.405,A -85,B 0,C 180,E1 -14925.43,E2 -14925.43} C_VEL
LIN {X 0,Y 326.77,Z 115.399,A -85,B 0,C 180,E1 -14928.835,E2 -14928.835} C_VEL
LIN {X 0,Y 326.924,Z 115.378,A -85,B 0,C 180,E1 -14932.585,E2 -14932.585} C_VEL
LIN {X 0,Y 326.769,Z 115.405,A -85,B 0,C 180,E1 -14935.061,E2 -14935.061} C_VEL
LIN {X 0,Y 327.043,Z 115.363,A -85,B 0,C 180,E1 -14937.533,E2 -14937.533} C_VEL
LIN {X 0,Y 327.166,Z 115.353,A -85,B 0,C 180,E1 -14939.996,E2 -14939.996} C_VEL
LIN {X 0,Y 327.049,Z 115.369,A -85,B 0,C 180,E1 -14942.459,E2 -14942.459} C_VEL
LIN {X 0,Y 326.934,Z 115.38,A -85,B 0,C 180,E1 -14946.495,E2 -14946.495} C_VEL
LIN {X 0,Y 326.787,Z 115.397,A -85,B 0,C 180,E1 -14949.903,E2 -14949.903} C_VEL
LIN {X 0,Y 326.761,Z 115.401,A -85,B 0,C 180,E1 -14953.681,E2 -14953.681} C_VEL
LIN {X 0,Y 326.699,Z 115.41,A -85,B 0,C 180,E1 -14957.523,E2 -14957.523} C_VEL
LIN {X 0,Y 326.661,Z 115.413,A -85,B 0,C 180,E1 -14960.13,E2 -14960.13} C_VEL
LIN {X 0,Y 326.646,Z 115.421,A -85,B 0,C 180,E1 -14964.124,E2 -14964.124} C_VEL
LIN {X 0,Y 326.67,Z 115.416,A -85,B 0,C 180,E1 -14966.853,E2 -14966.853} C_VEL
LIN {X 0,Y 326.605,Z 115.409,A -85,B 0,C 180,E1 -14970.598,E2 -14970.598} C_VEL
LIN {X 0,Y 326.597,Z 115.413,A -85,B 0,C 180,E1 -14974.014,E2 -14974.014} C_VEL
LIN {X 0,Y 326.615,Z 115.417,A -85,B 0,C 180,E1 -14977.233,E2 -14977.233} C_VEL
LIN {X 0,Y 326.605,Z 115.473,A -85,B 0,C 180,E1 -14979.117,E2 -14979.117} C_VEL
LIN {X 0,Y 328.475,Z 122.231,A -85,B 0,C 180,E1 -14981.543,E2 -14981.543} C_VEL
LIN {X 0,Y 338.134,Z 140.09,A -85,B 0,C 180,E1 -14983.259,E2 -14983.259} C_VEL
LIN {X 0,Y 345.804,Z 155.859,A -85,B 0,C 180,E1 -14984.564,E2 -14984.564} C_VEL
LIN {X 0,Y 347.889,Z 160.816,A -85,B 0,C 180,E1 -14984.92,E2 -14984.92} C_VEL
LIN {X 0,Y 344.682,Z 258.311,A -85,B 0,C 180,E1 -14987.007,E2 -14987.007} C_VEL
LIN {X 0,Y 343.708,Z 272.568,A -85,B 0,C 180,E1 -14987.533,E2 -14987.533} C_VEL
LIN {X 0,Y 342.395,Z 285.984,A -85,B 0,C 180,E1 -14988.254,E2 -14988.254} C_VEL
LIN {X 0,Y 340.975,Z 298.109,A -85,B 0,C 180,E1 -14989.123,E2 -14989.123} C_VEL
LIN {X 0,Y 339.178,Z 310.284,A -85,B 0,C 180,E1 -14990.225,E2 -14990.225} C_VEL
LIN {X 0,Y 337.003,Z 322.832,A -85,B 0,C 180,E1 -14991.651,E2 -14991.651} C_VEL
LIN {X 0,Y 334.837,Z 334.215,A -85,B 0,C 180,E1 -14993.264,E2 -14993.264} C_VEL
LIN {X 0,Y 332.958,Z 343.559,A -85,B 0,C 180,E1 -14994.885,E2 -14994.885} C_VEL
LIN {X 0,Y 330.964,Z 352.886,A -85,B 0,C 180,E1 -14996.851,E2 -14996.851} C_VEL
LIN {X 0,Y 329.236,Z 360.634,A -85,B 0,C 180,E1 -14998.859,E2 -14998.859} C_VEL
LIN {X 0,Y 327.736,Z 367.635,A -85,B 0,C 180,E1 -15001.122,E2 -15001.122} C_VEL
LIN {X 0,Y 326.721,Z 372.557,A -85,B 0,C 180,E1 -15003.144,E2 -15003.144} C_VEL
LIN {X 0,Y 326.039,Z 375.888,A -85,B 0,C 180,E1 -15004.855,E2 -15004.855} C_VEL
LIN {X 0,Y 325.392,Z 379.225,A -85,B 0,C 180,E1 -15007.12,E2 -15007.12} C_VEL
LIN {X 0,Y 325.118,Z 380.621,A -85,B 0,C 180,E1 -15008.438,E2 -15008.438} C_VEL
LIN {X 0,Y 324.757,Z 382.293,A -85,B 0,C 180,E1 -15011.056,E2 -15011.056} C_VEL
LIN {X 0,Y 324.723,Z 382.583,A -85,B 0,C 180,E1 -15012.36,E2 -15012.36} C_VEL
LIN {X 0,Y 324.631,Z 382.103,A -85,B 0,C 180,E1 -15014.941,E2 -15014.941} C_VEL
LIN {X 0,Y 324.804,Z 380.216,A -85,B 0,C 180,E1 -15017.502,E2 -15017.502} C_VEL
LIN {X 0,Y 325.056,Z 376.886,A -85,B 0,C 180,E1 -15020.038,E2 -15020.038} C_VEL
LIN {X 0,Y 325.517,Z 372.028,A -85,B 0,C 180,E1 -15022.555,E2 -15022.555} C_VEL
LIN {X 0,Y 325.989,Z 367.354,A -85,B 0,C 180,E1 -15024.431,E2 -15024.431} C_VEL
LIN {X 0,Y 326.815,Z 360.548,A -85,B 0,C 180,E1 -15026.608,E2 -15026.608} C_VEL
LIN {X 0,Y 327.942,Z 352.096,A -85,B 0,C 180,E1 -15028.77,E2 -15028.77} C_VEL
LIN {X 0,Y 329.196,Z 343.282,A -85,B 0,C 180,E1 -15030.61,E2 -15030.61} C_VEL
LIN {X 0,Y 330.628,Z 332.627,A -85,B 0,C 180,E1 -15032.435,E2 -15032.435} C_VEL
LIN {X 0,Y 331.982,Z 321.875,A -85,B 0,C 180,E1 -15033.943,E2 -15033.943} C_VEL
LIN {X 0,Y 333.435,Z 310.1,A -85,B 0,C 180,E1 -15035.289,E2 -15035.289} C_VEL
LIN {X 0,Y 334.778,Z 297.154,A -85,B 0,C 180,E1 -15036.477,E2 -15036.477} C_VEL
LIN {X 0,Y 335.937,Z 283.635,A -85,B 0,C 180,E1 -15037.436,E2 -15037.436} C_VEL
LIN {X 0,Y 336.855,Z 269.423,A -85,B 0,C 180,E1 -15038.17,E2 -15038.17} C_VEL
LIN {X 0,Y 337.41,Z 255.749,A -85,B 0,C 180,E1 -15038.646,E2 -15038.646} C_VEL
LIN {X 0,Y 339.976,Z 155.285,A -85,B 0,C 180,E1 -15040.774,E2 -15040.774} C_VEL
LIN {X 0,Y 338.442,Z 148.56,A -85,B 0,C 180,E1 -15041.036,E2 -15041.036} C_VEL
LIN {X 0,Y 329.65,Z 125.438,A -85,B 0,C 180,E1 -15042.227,E2 -15042.227} C_VEL
LIN {X 0,Y 327.97,Z 121.135,A -85,B 0,C 180,E1 -15042.49,E2 -15042.49} C_VEL
LIN {X 0,Y 326.775,Z 115.411,A -85,B 0,C 180,E1 -15044.188,E2 -15044.188} C_VEL
LIN {X 0,Y 326.679,Z 115.421,A -85,B 0,C 180,E1 -15047.527,E2 -15047.527} C_VEL
LIN {X 0,Y 326.66,Z 115.417,A -85,B 0,C 180,E1 -15049.751,E2 -15049.751} C_VEL
LIN {X 0,Y 325.972,Z 115.505,A -85,B 0,C 180,E1 -15050.78,E2 -15050.78} C_VEL
LIN {X 0,Y 323.099,Z 115.862,A -85,B 0,C 180,E1 -15052.456,E2 -15052.456} C_VEL
LIN {X 0,Y 320.684,Z 116.164,A -85,B 0,C 180,E1 -15053.814,E2 -15053.814} C_VEL
LIN {X 0,Y 319.663,Z 116.29,A -85,B 0,C 180,E1 -15054.865,E2 -15054.865} C_VEL
LIN {X 0,Y 319.587,Z 116.299,A -85,B 0,C 180,E1 -15055.221,E2 -15055.221} C_VEL
LIN {X 0,Y 319.556,Z 116.304,A -85,B 0,C 180,E1 -15058.935,E2 -15058.935} C_VEL
LIN {X 0,Y 319.506,Z 116.309,A -85,B 0,C 180,E1 -15061.862,E2 -15061.862} C_VEL
LIN {X 0,Y 319.574,Z 116.301,A -85,B 0,C 180,E1 -15065.551,E2 -15065.551} C_VEL
LIN {X 0,Y 319.603,Z 116.296,A -85,B 0,C 180,E1 -15068.001,E2 -15068.001} C_VEL
LIN {X 0,Y 319.617,Z 116.294,A -85,B 0,C 180,E1 -15071.624,E2 -15071.624} C_VEL
LIN {X 0,Y 319.623,Z 116.293,A -85,B 0,C 180,E1 -15075.289,E2 -15075.289} C_VEL
LIN {X 0,Y 319.555,Z 116.305,A -85,B 0,C 180,E1 -15078.723,E2 -15078.723} C_VEL
LIN {X 0,Y 319.572,Z 116.297,A -85,B 0,C 180,E1 -15082.342,E2 -15082.342} C_VEL
LIN {X 0,Y 319.534,Z 116.304,A -85,B 0,C 180,E1 -15085.127,E2 -15085.127} C_VEL
LIN {X 0,Y 319.55,Z 116.3,A -85,B 0,C 180,E1 -15089.06,E2 -15089.06} C_VEL
LIN {X 0,Y 319.587,Z 116.297,A -85,B 0,C 180,E1 -15092.502,E2 -15092.502} C_VEL
LIN {X 0,Y 319.605,Z 116.295,A -85,B 0,C 180,E1 -15095.31,E2 -15095.31} C_VEL
LIN {X 0,Y 319.621,Z 116.298,A -85,B 0,C 180,E1 -15098.055,E2 -15098.055} C_VEL
LIN {X 0,Y 319.687,Z 116.285,A -85,B 0,C 180,E1 -15100.957,E2 -15100.957} C_VEL
LIN {X 0,Y 319.714,Z 116.282,A -85,B 0,C 180,E1 -15105.28,E2 -15105.28} C_VEL
LIN {X 0,Y 319.744,Z 116.28,A -85,B 0,C 180,E1 -15109.877,E2 -15109.877} C_VEL
LIN {X 0,Y 319.919,Z 116.251,A -85,B 0,C 180,E1 -15112.43,E2 -15112.43} C_VEL
LIN {X 0,Y 319.739,Z 116.274,A -85,B 0,C 180,E1 -15114.96,E2 -15114.96} C_VEL
LIN {X 0,Y 319.998,Z 116.251,A -85,B 0,C 180,E1 -15117.487,E2 -15117.487} C_VEL
LIN {X 0,Y 320.159,Z 116.227,A -85,B 0,C 180,E1 -15120.004,E2 -15120.004} C_VEL
LIN {X 0,Y 319.982,Z 116.246,A -85,B 0,C 180,E1 -15122.522,E2 -15122.522} C_VEL
LIN {X 0,Y 319.943,Z 116.25,A -85,B 0,C 180,E1 -15126.31,E2 -15126.31} C_VEL
LIN {X 0,Y 319.835,Z 116.27,A -85,B 0,C 180,E1 -15128.852,E2 -15128.852} C_VEL
LIN {X 0,Y 319.675,Z 116.289,A -85,B 0,C 180,E1 -15132.704,E2 -15132.704} C_VEL
LIN {X 0,Y 319.694,Z 116.286,A -85,B 0,C 180,E1 -15135.3,E2 -15135.3} C_VEL
LIN {X 0,Y 319.671,Z 116.289,A -85,B 0,C 180,E1 -15139.259,E2 -15139.259} C_VEL
LIN {X 0,Y 319.567,Z 116.301,A -85,B 0,C 180,E1 -15143.323,E2 -15143.323} C_VEL
LIN {X 0,Y 319.632,Z 116.294,A -85,B 0,C 180,E1 -15146.092,E2 -15146.092} C_VEL
LIN {X 0,Y 319.588,Z 116.299,A -85,B 0,C 180,E1 -15148.937,E2 -15148.937} C_VEL
LIN {X 0,Y 319.531,Z 116.305,A -85,B 0,C 180,E1 -15151.866,E2 -15151.866} C_VEL
LIN {X 0,Y 319.579,Z 116.299,A -85,B 0,C 180,E1 -15155.546,E2 -15155.546} C_VEL
LIN {X 0,Y 319.573,Z 116.304,A -85,B 0,C 180,E1 -15158.012,E2 -15158.012} C_VEL
LIN {X 0,Y 319.527,Z 116.305,A -85,B 0,C 180,E1 -15161.6,E2 -15161.6} C_VEL
LIN {X 0,Y 319.49,Z 116.312,A -85,B 0,C 180,E1 -15165.26,E2 -15165.26} C_VEL
LIN {X 0,Y 319.531,Z 116.304,A -85,B 0,C 180,E1 -15168.715,E2 -15168.715} C_VEL
LIN {X 0,Y 319.565,Z 116.305,A -85,B 0,C 180,E1 -15172.351,E2 -15172.351} C_VEL
LIN {X 0,Y 319.599,Z 116.347,A -85,B 0,C 180,E1 -15175.705,E2 -15175.705} C_VEL
LIN {X 0,Y 322.51,Z 129.116,A -85,B 0,C 180,E1 -15179.198,E2 -15179.198} C_VEL
LIN {X 0,Y 324.192,Z 137.053,A -85,B 0,C 180,E1 -15181.26,E2 -15181.26} C_VEL
LIN {X 0,Y 327.536,Z 146.751,A -85,B 0,C 180,E1 -15181.753,E2 -15181.753} C_VEL
LIN {X 0,Y 332.949,Z 181.321,A -85,B 0,C 180,E1 -15182.965,E2 -15182.965} C_VEL
LIN {X 0,Y 330.609,Z 275.166,A -85,B 0,C 180,E1 -15185.01,E2 -15185.01} C_VEL
LIN {X 0,Y 329.797,Z 289.035,A -85,B 0,C 180,E1 -15185.532,E2 -15185.532} C_VEL
LIN {X 0,Y 328.643,Z 302.67,A -85,B 0,C 180,E1 -15186.28,E2 -15186.28} C_VEL
LIN {X 0,Y 327.35,Z 315.977,A -85,B 0,C 180,E1 -15187.268,E2 -15187.268} C_VEL
LIN {X 0,Y 325.811,Z 328.807,A -85,B 0,C 180,E1 -15188.49,E2 -15188.49} C_VEL
LIN {X 0,Y 324.337,Z 340.491,A -85,B 0,C 180,E1 -15189.882,E2 -15189.882} C_VEL
LIN {X 0,Y 322.929,Z 350.19,A -85,B 0,C 180,E1 -15191.278,E2 -15191.278} C_VEL
LIN {X 0,Y 321.439,Z 360.963,A -85,B 0,C 180,E1 -15193.162,E2 -15193.162} C_VEL
LIN {X 0,Y 320.223,Z 370.07,A -85,B 0,C 180,E1 -15195.112,E2 -15195.112} C_VEL
LIN {X 0,Y 319.275,Z 378.339,A -85,B 0,C 180,E1 -15197.286,E2 -15197.286} C_VEL
LIN {X 0,Y 318.528,Z 384.23,A -85,B 0,C 180,E1 -15199.192,E2 -15199.192} C_VEL
LIN {X 0,Y 318.137,Z 389.08,A -85,B 0,C 180,E1 -15201.106,E2 -15201.106} C_VEL
LIN {X 0,Y 317.899,Z 392.998,A -85,B 0,C 180,E1 -15203.018,E2 -15203.018} C_VEL
LIN {X 0,Y 317.759,Z 395.989,A -85,B 0,C 180,E1 -15204.926,E2 -15204.926} C_VEL
LIN {X 0,Y 317.787,Z 397.539,A -85,B 0,C 180,E1 -15206.198,E2 -15206.198} C_VEL
LIN {X 0,Y 317.748,Z 399.578,A -85,B 0,C 180,E1 -15208.734,E2 -15208.734} C_VEL
LIN {X 0,Y 317.786,Z 400.087,A -85,B 0,C 180,E1 -15210.002,E2 -15210.002} C_VEL
LIN {X 0,Y 317.753,Z 400.088,A -85,B 0,C 180,E1 -15212.537,E2 -15212.537} C_VEL
LIN {X 0,Y 317.786,Z 398.755,A -85,B 0,C 180,E1 -15215.077,E2 -15215.077} C_VEL
LIN {X 0,Y 318.034,Z 396.068,A -85,B 0,C 180,E1 -15217.621,E2 -15217.621} C_VEL
LIN {X 0,Y 318.583,Z 391.965,A -85,B 0,C 180,E1 -15220.167,E2 -15220.167} C_VEL
LIN {X 0,Y 319.619,Z 386.336,A -85,B 0,C 180,E1 -15222.704,E2 -15222.704} C_VEL
LIN {X 0,Y 320.858,Z 380.026,A -85,B 0,C 180,E1 -15224.916,E2 -15224.916} C_VEL
LIN {X 0,Y 322.477,Z 372.211,A -85,B 0,C 180,E1 -15227.112,E2 -15227.112} C_VEL
LIN {X 0,Y 324.304,Z 364.076,A -85,B 0,C 180,E1 -15228.971,E2 -15228.971} C_VEL
LIN {X 0,Y 326.462,Z 354.308,A -85,B 0,C 180,E1 -15230.808,E2 -15230.808} C_VEL
LIN {X 0,Y 328.763,Z 343.491,A -85,B 0,C 180,E1 -15232.467,E2 -15232.467} C_VEL
LIN {X 0,Y 330.964,Z 332.069,A -85,B 0,C 180,E1 -15233.894,E2 -15233.894} C_VEL
LIN {X 0,Y 333.063,Z 319.782,A -85,B 0,C 180,E1 -15235.131,E2 -15235.131} C_VEL
LIN {X 0,Y 334.933,Z 306.949,A -85,B 0,C 180,E1 -15236.147,E2 -15236.147} C_VEL
LIN {X 0,Y 336.632,Z 293.077,A -85,B 0,C 180,E1 -15236.966,E2 -15236.966} C_VEL
LIN {X 0,Y 337.955,Z 278.45,A -85,B 0,C 180,E1 -15237.563,E2 -15237.563} C_VEL
LIN {X 0,Y 338.685,Z 263.036,A -85,B 0,C 180,E1 -15237.961,E2 -15237.961} C_VEL
LIN {X 0,Y 341.188,Z 183.125,A -85,B 0,C 180,E1 -15239.697,E2 -15239.697} C_VEL
LIN {X 0,Y 337.028,Z 161.159,A -85,B 0,C 180,E1 -15240.75,E2 -15240.75} C_VEL
LIN {X 0,Y 331.316,Z 148.457,A -85,B 0,C 180,E1 -15241.793,E2 -15241.793} C_VEL
LIN {X 0,Y 326.487,Z 139.186,A -85,B 0,C 180,E1 -15242.68,E2 -15242.68} C_VEL
LIN {X 0,Y 324.945,Z 135.844,A -85,B 0,C 180,E1 -15243.029,E2 -15243.029} C_VEL
LIN {X 0,Y 322.363,Z 125.931,A -85,B 0,C 180,E1 -15246.225,E2 -15246.225} C_VEL
LIN {X 0,Y 319.564,Z 116.296,A -85,B 0,C 180,E1 -15249.666,E2 -15249.666} C_VEL
LIN {X 0,Y 319.537,Z 116.306,A -85,B 0,C 180,E1 -15253.46,E2 -15253.46} C_VEL
LIN {X 0,Y 319.569,Z 116.299,A -85,B 0,C 180,E1 -15257.015,E2 -15257.015} C_VEL
LIN {X 0,Y 319.561,Z 116.296,A -85,B 0,C 180,E1 -15260.369,E2 -15260.369} C_VEL
LIN {X 0,Y 319.594,Z 116.3,A -85,B 0,C 180,E1 -15264.456,E2 -15264.456} C_VEL
LIN {X 0,Y 319.539,Z 116.303,A -85,B 0,C 180,E1 -15268.135,E2 -15268.135} C_VEL
LIN {X 0,Y 319.587,Z 116.295,A -85,B 0,C 180,E1 -15271.601,E2 -15271.601} C_VEL
LIN {X 0,Y 319.589,Z 116.294,A -85,B 0,C 180,E1 -15275.299,E2 -15275.299} C_VEL
LIN {X 0,Y 319.614,Z 116.288,A -85,B 0,C 180,E1 -15279.397,E2 -15279.397} C_VEL
LIN {X 0,Y 319.672,Z 116.29,A -85,B 0,C 180,E1 -15282.07,E2 -15282.07} C_VEL
LIN {X 0,Y 319.745,Z 116.281,A -85,B 0,C 180,E1 -15286.005,E2 -15286.005} C_VEL
LIN {X 0,Y 319.747,Z 116.279,A -85,B 0,C 180,E1 -15289.869,E2 -15289.869} C_VEL
LIN {X 0,Y 319.912,Z 116.256,A -85,B 0,C 180,E1 -15293.69,E2 -15293.69} C_VEL
LIN {X 0,Y 319.986,Z 116.242,A -85,B 0,C 180,E1 -15297.478,E2 -15297.478} C_VEL
LIN {X 0,Y 320.119,Z 116.231,A -85,B 0,C 180,E1 -15299.996,E2 -15299.996} C_VEL
LIN {X 0,Y 319.992,Z 116.249,A -85,B 0,C 180,E1 -15302.513,E2 -15302.513} C_VEL
LIN {X 0,Y 319.9,Z 116.257,A -85,B 0,C 180,E1 -15306.48,E2 -15306.48} C_VEL
LIN {X 0,Y 319.739,Z 116.276,A -85,B 0,C 180,E1 -15310.123,E2 -15310.123} C_VEL
LIN {X 0,Y 319.734,Z 116.278,A -85,B 0,C 180,E1 -15313.987,E2 -15313.987} C_VEL
LIN {X 0,Y 319.658,Z 116.291,A -85,B 0,C 180,E1 -15317.922,E2 -15317.922} C_VEL
LIN {X 0,Y 319.612,Z 116.292,A -85,B 0,C 180,E1 -15320.594,E2 -15320.594} C_VEL
LIN {X 0,Y 319.566,Z 116.299,A -85,B 0,C 180,E1 -15323.314,E2 -15323.314} C_VEL
LIN {X 0,Y 319.61,Z 116.292,A -85,B 0,C 180,E1 -15326.085,E2 -15326.085} C_VEL
LIN {X 0,Y 319.561,Z 116.289,A -85,B 0,C 180,E1 -15328.931,E2 -15328.931} C_VEL
LIN {X 0,Y 319.516,Z 116.311,A -85,B 0,C 180,E1 -15331.857,E2 -15331.857} C_VEL
LIN {X 0,Y 319.569,Z 116.299,A -85,B 0,C 180,E1 -15335.538,E2 -15335.538} C_VEL
LIN {X 0,Y 319.567,Z 116.479,A -85,B 0,C 180,E1 -15338.302,E2 -15338.302} C_VEL
LIN {X 0,Y 321.311,Z 122.501,A -85,B 0,C 180,E1 -15340.552,E2 -15340.552} C_VEL
LIN {X 0,Y 323.673,Z 126.67,A -85,B 0,C 180,E1 -15341.005,E2 -15341.005} C_VEL
LIN {X 0,Y 332.426,Z 142.686,A -85,B 0,C 180,E1 -15342.617,E2 -15342.617} C_VEL
LIN {X 0,Y 340.714,Z 159.875,A -85,B 0,C 180,E1 -15344.078,E2 -15344.078} C_VEL
LIN {X 0,Y 341.906,Z 162.697,A -85,B 0,C 180,E1 -15344.289,E2 -15344.289} C_VEL
LIN {X 0,Y 338.642,Z 258.879,A -85,B 0,C 180,E1 -15346.393,E2 -15346.393} C_VEL
LIN {X 0,Y 337.559,Z 273.684,A -85,B 0,C 180,E1 -15346.958,E2 -15346.958} C_VEL
LIN {X 0,Y 336.015,Z 288.309,A -85,B 0,C 180,E1 -15347.783,E2 -15347.783} C_VEL
LIN {X 0,Y 334.422,Z 300.916,A -85,B 0,C 180,E1 -15348.747,E2 -15348.747} C_VEL
LIN {X 0,Y 332.512,Z 312.853,A -85,B 0,C 180,E1 -15349.894,E2 -15349.894} C_VEL
LIN {X 0,Y 330.333,Z 324.759,A -85,B 0,C 180,E1 -15351.318,E2 -15351.318} C_VEL
LIN {X 0,Y 328.23,Z 335.195,A -85,B 0,C 180,E1 -15352.857,E2 -15352.857} C_VEL
LIN {X 0,Y 326.099,Z 345.121,A -85,B 0,C 180,E1 -15354.642,E2 -15354.642} C_VEL
LIN {X 0,Y 323.897,Z 354.713,A -85,B 0,C 180,E1 -15356.776,E2 -15356.776} C_VEL
LIN {X 0,Y 322.191,Z 362.053,A -85,B 0,C 180,E1 -15358.796,E2 -15358.796} C_VEL
LIN {X 0,Y 320.637,Z 368.917,A -85,B 0,C 180,E1 -15361.168,E2 -15361.168} C_VEL
LIN {X 0,Y 319.603,Z 373.583,A -85,B 0,C 180,E1 -15363.204,E2 -15363.204} C_VEL
LIN {X 0,Y 318.84,Z 377.208,A -85,B 0,C 180,E1 -15365.239,E2 -15365.239} C_VEL
LIN {X 0,Y 318.42,Z 379.104,A -85,B 0,C 180,E1 -15366.59,E2 -15366.59} C_VEL
LIN {X 0,Y 318.129,Z 380.703,A -85,B 0,C 180,E1 -15368.086,E2 -15368.086} C_VEL
LIN {X 0,Y 317.711,Z 382.391,A -85,B 0,C 180,E1 -15370.619,E2 -15370.619} C_VEL
LIN {X 0,Y 317.575,Z 382.754,A -85,B 0,C 180,E1 -15373.278,E2 -15373.278} C_VEL
LIN {X 0,Y 317.587,Z 381.704,A -85,B 0,C 180,E1 -15375.91,E2 -15375.91} C_VEL
LIN {X 0,Y 317.694,Z 380.652,A -85,B 0,C 180,E1 -15377.218,E2 -15377.218} C_VEL
LIN {X 0,Y 317.912,Z 377.491,A -85,B 0,C 180,E1 -15379.812,E2 -15379.812} C_VEL
LIN {X 0,Y 318.252,Z 374.107,A -85,B 0,C 180,E1 -15381.745,E2 -15381.745} C_VEL
LIN {X 0,Y 318.872,Z 368.232,A -85,B 0,C 180,E1 -15384.306,E2 -15384.306} C_VEL
LIN {X 0,Y 319.672,Z 361.621,A -85,B 0,C 180,E1 -15386.532,E2 -15386.532} C_VEL
LIN {X 0,Y 320.839,Z 353.405,A -85,B 0,C 180,E1 -15388.743,E2 -15388.743} C_VEL
LIN {X 0,Y 322.089,Z 344.817,A -85,B 0,C 180,E1 -15390.623,E2 -15390.623} C_VEL
LIN {X 0,Y 323.571,Z 334.111,A -85,B 0,C 180,E1 -15392.539,E2 -15392.539} C_VEL
LIN {X 0,Y 325.052,Z 322.829,A -85,B 0,C 180,E1 -15394.183,E2 -15394.183} C_VEL
LIN {X 0,Y 326.539,Z 311.215,A -85,B 0,C 180,E1 -15395.556,E2 -15395.556} C_VEL
LIN {X 0,Y 327.925,Z 298.475,A -85,B 0,C 180,E1 -15396.768,E2 -15396.768} C_VEL
LIN {X 0,Y 329.137,Z 285.274,A -85,B 0,C 180,E1 -15397.745,E2 -15397.745} C_VEL
LIN {X 0,Y 330.122,Z 270.973,A -85,B 0,C 180,E1 -15398.53,E2 -15398.53} C_VEL
LIN {X 0,Y 330.751,Z 256.707,A -85,B 0,C 180,E1 -15399.053,E2 -15399.053} C_VEL
LIN {X 0,Y 333.455,Z 156.581,A -85,B 0,C 180,E1 -15401.21,E2 -15401.21} C_VEL
LIN {X 0,Y 332.252,Z 151.142,A -85,B 0,C 180,E1 -15401.425,E2 -15401.425} C_VEL
LIN {X 0,Y 323.226,Z 127.36,A -85,B 0,C 180,E1 -15402.688,E2 -15402.688} C_VEL
LIN {X 0,Y 320.82,Z 121.387,A -85,B 0,C 180,E1 -15403.044,E2 -15403.044} C_VEL
LIN {X 0,Y 319.701,Z 116.292,A -85,B 0,C 180,E1 -15404.603,E2 -15404.603} C_VEL
LIN {X 0,Y 319.633,Z 116.297,A -85,B 0,C 180,E1 -15407.926,E2 -15407.926} C_VEL
LIN {X 0,Y 319.604,Z 116.297,A -85,B 0,C 180,E1 -15410.598,E2 -15410.598} C_VEL
LIN {X 0,Y 319.604,Z 116.301,A -85,B 0,C 180,E1 -15413.315,E2 -15413.315} C_VEL
LIN {X 0,Y 319.587,Z 116.299,A -85,B 0,C 180,E1 -15415.221,E2 -15415.221} C_VEL
LIN {X 0,Y 318.927,Z 116.382,A -85,B 0,C 180,E1 -15416.273,E2 -15416.273} C_VEL
LIN {X 0,Y 316.036,Z 116.74,A -85,B 0,C 180,E1 -15417.985,E2 -15417.985} C_VEL
LIN {X 0,Y 313.587,Z 117.05,A -85,B 0,C 180,E1 -15419.372,E2 -15419.372} C_VEL
LIN {X 0,Y 312.554,Z 117.175,A -85,B 0,C 180,E1 -15420.448,E2 -15420.448} C_VEL
LIN {X 0,Y 312.48,Z 117.185,A -85,B 0,C 180,E1 -15420.812,E2 -15420.812} C_VEL
LIN {X 0,Y 312.484,Z 117.183,A -85,B 0,C 180,E1 -15424.21,E2 -15424.21} C_VEL
LIN {X 0,Y 312.576,Z 117.171,A -85,B 0,C 180,E1 -15428.109,E2 -15428.109} C_VEL
LIN {X 0,Y 312.552,Z 117.173,A -85,B 0,C 180,E1 -15432.104,E2 -15432.104} C_VEL
LIN {X 0,Y 312.567,Z 117.171,A -85,B 0,C 180,E1 -15436.011,E2 -15436.011} C_VEL
LIN {X 0,Y 312.519,Z 117.176,A -85,B 0,C 180,E1 -15439.868,E2 -15439.868} C_VEL
LIN {X 0,Y 312.526,Z 117.175,A -85,B 0,C 180,E1 -15442.622,E2 -15442.622} C_VEL
LIN {X 0,Y 312.494,Z 117.185,A -85,B 0,C 180,E1 -15446.314,E2 -15446.314} C_VEL
LIN {X 0,Y 312.523,Z 117.174,A -85,B 0,C 180,E1 -15450.354,E2 -15450.354} C_VEL
LIN {X 0,Y 312.583,Z 117.17,A -85,B 0,C 180,E1 -15454.067,E2 -15454.067} C_VEL
LIN {X 0,Y 312.601,Z 117.17,A -85,B 0,C 180,E1 -15457.535,E2 -15457.535} C_VEL
LIN {X 0,Y 312.626,Z 117.167,A -85,B 0,C 180,E1 -15461.661,E2 -15461.661} C_VEL
LIN {X 0,Y 312.677,Z 117.161,A -85,B 0,C 180,E1 -15465.69,E2 -15465.69} C_VEL
LIN {X 0,Y 312.689,Z 117.161,A -85,B 0,C 180,E1 -15469.646,E2 -15469.646} C_VEL
LIN {X 0,Y 312.858,Z 117.13,A -85,B 0,C 180,E1 -15472.258,E2 -15472.258} C_VEL
LIN {X 0,Y 312.709,Z 117.148,A -85,B 0,C 180,E1 -15474.847,E2 -15474.847} C_VEL
LIN {X 0,Y 312.942,Z 117.128,A -85,B 0,C 180,E1 -15477.43,E2 -15477.43} C_VEL
LIN {X 0,Y 313.111,Z 117.105,A -85,B 0,C 180,E1 -15480.004,E2 -15480.004} C_VEL
LIN {X 0,Y 312.929,Z 117.125,A -85,B 0,C 180,E1 -15482.579,E2 -15482.579} C_VEL
LIN {X 0,Y 312.902,Z 117.126,A -85,B 0,C 180,E1 -15486.452,E2 -15486.452} C_VEL
LIN {X 0,Y 312.78,Z 117.15,A -85,B 0,C 180,E1 -15489.053,E2 -15489.053} C_VEL
LIN {X 0,Y 312.628,Z 117.168,A -85,B 0,C 180,E1 -15492.995,E2 -15492.995} C_VEL
LIN {X 0,Y 312.633,Z 117.164,A -85,B 0,C 180,E1 -15495.654,E2 -15495.654} C_VEL
LIN {X 0,Y 312.627,Z 117.167,A -85,B 0,C 180,E1 -15499.241,E2 -15499.241} C_VEL
LIN {X 0,Y 312.543,Z 117.179,A -85,B 0,C 180,E1 -15502.793,E2 -15502.793} C_VEL
LIN {X 0,Y 312.6,Z 117.169,A -85,B 0,C 180,E1 -15505.939,E2 -15505.939} C_VEL
LIN {X 0,Y 312.544,Z 117.175,A -85,B 0,C 180,E1 -15509.654,E2 -15509.654} C_VEL
LIN {X 0,Y 312.519,Z 117.178,A -85,B 0,C 180,E1 -15513.692,E2 -15513.692} C_VEL
LIN {X 0,Y 312.526,Z 117.178,A -85,B 0,C 180,E1 -15517.389,E2 -15517.389} C_VEL
LIN {X 0,Y 312.491,Z 117.181,A -85,B 0,C 180,E1 -15520.713,E2 -15520.713} C_VEL
LIN {X 0,Y 312.453,Z 117.191,A -85,B 0,C 180,E1 -15524.213,E2 -15524.213} C_VEL
LIN {X 0,Y 312.487,Z 117.185,A -85,B 0,C 180,E1 -15527.922,E2 -15527.922} C_VEL
LIN {X 0,Y 312.506,Z 117.182,A -85,B 0,C 180,E1 -15530.975,E2 -15530.975} C_VEL
LIN {X 0,Y 312.539,Z 117.182,A -85,B 0,C 180,E1 -15535.014,E2 -15535.014} C_VEL
LIN {X 0,Y 312.58,Z 117.423,A -85,B 0,C 180,E1 -15535.313,E2 -15535.313} C_VEL
LIN {X 0,Y 315.764,Z 131.334,A -85,B 0,C 180,E1 -15539.211,E2 -15539.211} C_VEL
LIN {X 0,Y 316.911,Z 136.947,A -85,B 0,C 180,E1 -15540.672,E2 -15540.672} C_VEL
LIN {X 0,Y 321.222,Z 148.945,A -85,B 0,C 180,E1 -15541.312,E2 -15541.312} C_VEL
LIN {X 0,Y 326.397,Z 182.948,A -85,B 0,C 180,E1 -15542.527,E2 -15542.527} C_VEL
LIN {X 0,Y 324.007,Z 274.297,A -85,B 0,C 180,E1 -15544.55,E2 -15544.55} C_VEL
LIN {X 0,Y 323.167,Z 288.423,A -85,B 0,C 180,E1 -15545.082,E2 -15545.082} C_VEL
LIN {X 0,Y 321.957,Z 302.166,A -85,B 0,C 180,E1 -15545.842,E2 -15545.842} C_VEL
LIN {X 0,Y 320.607,Z 315.669,A -85,B 0,C 180,E1 -15546.859,E2 -15546.859} C_VEL
LIN {X 0,Y 319.17,Z 327.716,A -85,B 0,C 180,E1 -15548.019,E2 -15548.019} C_VEL
LIN {X 0,Y 317.739,Z 338.366,A -85,B 0,C 180,E1 -15549.276,E2 -15549.276} C_VEL
LIN {X 0,Y 316.103,Z 349.385,A -85,B 0,C 180,E1 -15550.858,E2 -15550.858} C_VEL
LIN {X 0,Y 314.555,Z 360.267,A -85,B 0,C 180,E1 -15552.782,E2 -15552.782} C_VEL
LIN {X 0,Y 313.372,Z 369,A -85,B 0,C 180,E1 -15554.666,E2 -15554.666} C_VEL
LIN {X 0,Y 312.383,Z 376.674,A -85,B 0,C 180,E1 -15556.669,E2 -15556.669} C_VEL
LIN {X 0,Y 311.493,Z 383.763,A -85,B 0,C 180,E1 -15558.945,E2 -15558.945} C_VEL
LIN {X 0,Y 311.09,Z 388.673,A -85,B 0,C 180,E1 -15560.903,E2 -15560.903} C_VEL
LIN {X 0,Y 310.817,Z 392.642,A -85,B 0,C 180,E1 -15562.858,E2 -15562.858} C_VEL
LIN {X 0,Y 310.675,Z 395.661,A -85,B 0,C 180,E1 -15564.81,E2 -15564.81} C_VEL
LIN {X 0,Y 310.697,Z 397.236,A -85,B 0,C 180,E1 -15566.111,E2 -15566.111} C_VEL
LIN {X 0,Y 310.662,Z 399.324,A -85,B 0,C 180,E1 -15568.706,E2 -15568.706} C_VEL
LIN {X 0,Y 310.696,Z 399.855,A -85,B 0,C 180,E1 -15570.002,E2 -15570.002} C_VEL
LIN {X 0,Y 310.676,Z 399.908,A -85,B 0,C 180,E1 -15572.595,E2 -15572.595} C_VEL
LIN {X 0,Y 310.697,Z 398.629,A -85,B 0,C 180,E1 -15575.193,E2 -15575.193} C_VEL
LIN {X 0,Y 310.982,Z 396.004,A -85,B 0,C 180,E1 -15577.795,E2 -15577.795} C_VEL
LIN {X 0,Y 311.561,Z 391.959,A -85,B 0,C 180,E1 -15580.398,E2 -15580.398} C_VEL
LIN {X 0,Y 312.653,Z 386.391,A -85,B 0,C 180,E1 -15582.992,E2 -15582.992} C_VEL
LIN {X 0,Y 313.985,Z 380.144,A -85,B 0,C 180,E1 -15585.25,E2 -15585.25} C_VEL
LIN {X 0,Y 315.671,Z 372.398,A -85,B 0,C 180,E1 -15587.493,E2 -15587.493} C_VEL
LIN {X 0,Y 317.903,Z 362.864,A -85,B 0,C 180,E1 -15589.704,E2 -15589.704} C_VEL
LIN {X 0,Y 320.228,Z 352.895,A -85,B 0,C 180,E1 -15591.57,E2 -15591.57} C_VEL
LIN {X 0,Y 322.679,Z 341.825,A -85,B 0,C 180,E1 -15593.253,E2 -15593.253} C_VEL
LIN {X 0,Y 324.96,Z 330.304,A -85,B 0,C 180,E1 -15594.675,E2 -15594.675} C_VEL
LIN {X 0,Y 327.258,Z 317.291,A -85,B 0,C 180,E1 -15595.95,E2 -15595.95} C_VEL
LIN {X 0,Y 329.177,Z 303.789,A -85,B 0,C 180,E1 -15596.983,E2 -15596.983} C_VEL
LIN {X 0,Y 330.961,Z 289.599,A -85,B 0,C 180,E1 -15597.767,E2 -15597.767} C_VEL
LIN {X 0,Y 332.171,Z 275.629,A -85,B 0,C 180,E1 -15598.3,E2 -15598.3} C_VEL
LIN {X 0,Y 333.394,Z 243.657,A -85,B 0,C 180,E1 -15599.04,E2 -15599.04} C_VEL
LIN {X 0,Y 335.301,Z 184.12,A -85,B 0,C 180,E1 -15600.359,E2 -15600.359} C_VEL
LIN {X 0,Y 331.522,Z 163.92,A -85,B 0,C 180,E1 -15601.354,E2 -15601.354} C_VEL
LIN {X 0,Y 325.35,Z 150.491,A -85,B 0,C 180,E1 -15602.521,E2 -15602.521} C_VEL
LIN {X 0,Y 319.302,Z 139.073,A -85,B 0,C 180,E1 -15603.684,E2 -15603.684} C_VEL
LIN {X 0,Y 317.676,Z 135.611,A -85,B 0,C 180,E1 -15604.057,E2 -15604.057} C_VEL
LIN {X 0,Y 315.342,Z 126.886,A -85,B 0,C 180,E1 -15606.997,E2 -15606.997} C_VEL
LIN {X 0,Y 313.171,Z 119.385,A -85,B 0,C 180,E1 -15609.714,E2 -15609.714} C_VEL
LIN {X 0,Y 312.48,Z 117.174,A -85,B 0,C 180,E1 -15610.625,E2 -15610.625} C_VEL
LIN {X 0,Y 312.467,Z 117.191,A -85,B 0,C 180,E1 -15614.209,E2 -15614.209} C_VEL
LIN {X 0,Y 312.483,Z 117.167,A -85,B 0,C 180,E1 -15617.921,E2 -15617.921} C_VEL
LIN {X 0,Y 312.511,Z 117.182,A -85,B 0,C 180,E1 -15620.969,E2 -15620.969} C_VEL
LIN {X 0,Y 312.545,Z 117.178,A -85,B 0,C 180,E1 -15624.218,E2 -15624.218} C_VEL
LIN {X 0,Y 312.517,Z 117.184,A -85,B 0,C 180,E1 -15627.332,E2 -15627.332} C_VEL
LIN {X 0,Y 312.522,Z 117.178,A -85,B 0,C 180,E1 -15631.29,E2 -15631.29} C_VEL
LIN {X 0,Y 312.563,Z 117.176,A -85,B 0,C 180,E1 -15634.705,E2 -15634.705} C_VEL
LIN {X 0,Y 312.578,Z 117.175,A -85,B 0,C 180,E1 -15637.524,E2 -15637.524} C_VEL
LIN {X 0,Y 312.652,Z 117.165,A -85,B 0,C 180,E1 -15641.653,E2 -15641.653} C_VEL
LIN {X 0,Y 312.707,Z 117.157,A -85,B 0,C 180,E1 -15645.683,E2 -15645.683} C_VEL
LIN {X 0,Y 312.697,Z 117.157,A -85,B 0,C 180,E1 -15649.638,E2 -15649.638} C_VEL
LIN {X 0,Y 312.807,Z 117.136,A -85,B 0,C 180,E1 -15652.249,E2 -15652.249} C_VEL
LIN {X 0,Y 312.707,Z 117.158,A -85,B 0,C 180,E1 -15654.838,E2 -15654.838} C_VEL
LIN {X 0,Y 312.992,Z 117.123,A -85,B 0,C 180,E1 -15658.709,E2 -15658.709} C_VEL
LIN {X 0,Y 312.992,Z 117.11,A -85,B 0,C 180,E1 -15661.282,E2 -15661.282} C_VEL
LIN {X 0,Y 312.707,Z 117.148,A -85,B 0,C 180,E1 -15665.153,E2 -15665.153} C_VEL
LIN {X 0,Y 312.822,Z 117.145,A -85,B 0,C 180,E1 -15667.742,E2 -15667.742} C_VEL
LIN {X 0,Y 312.666,Z 117.164,A -85,B 0,C 180,E1 -15671.667,E2 -15671.667} C_VEL
LIN {X 0,Y 312.702,Z 117.158,A -85,B 0,C 180,E1 -15674.883,E2 -15674.883} C_VEL
LIN {X 0,Y 312.629,Z 117.165,A -85,B 0,C 180,E1 -15679.231,E2 -15679.231} C_VEL
LIN {X 0,Y 312.542,Z 117.175,A -85,B 0,C 180,E1 -15682.783,E2 -15682.783} C_VEL
LIN {X 0,Y 312.59,Z 117.167,A -85,B 0,C 180,E1 -15685.927,E2 -15685.927} C_VEL
LIN {X 0,Y 312.501,Z 117.162,A -85,B 0,C 180,E1 -15689.649,E2 -15689.649} C_VEL
LIN {X 0,Y 312.51,Z 117.168,A -85,B 0,C 180,E1 -15693.683,E2 -15693.683} C_VEL
LIN {X 0,Y 312.533,Z 117.33,A -85,B 0,C 180,E1 -15697.377,E2 -15697.377} C_VEL
LIN {X 0,Y 314.132,Z 122.959,A -85,B 0,C 180,E1 -15699.504,E2 -15699.504} C_VEL
LIN {X 0,Y 322.036,Z 136.608,A -85,B 0,C 180,E1 -15701.058,E2 -15701.058} C_VEL
LIN {X 0,Y 329.36,Z 150.512,A -85,B 0,C 180,E1 -15702.433,E2 -15702.433} C_VEL
LIN {X 0,Y 336.002,Z 164.718,A -85,B 0,C 180,E1 -15703.642,E2 -15703.642} C_VEL
LIN {X 0,Y 332.666,Z 259.257,A -85,B 0,C 180,E1 -15705.745,E2 -15705.745} C_VEL
LIN {X 0,Y 331.559,Z 273.78,A -85,B 0,C 180,E1 -15706.307,E2 -15706.307} C_VEL
LIN {X 0,Y 329.962,Z 288.315,A -85,B 0,C 180,E1 -15707.135,E2 -15707.135} C_VEL
LIN {X 0,Y 328.163,Z 301.893,A -85,B 0,C 180,E1 -15708.194,E2 -15708.194} C_VEL
LIN {X 0,Y 326.109,Z 314.087,A -85,B 0,C 180,E1 -15709.404,E2 -15709.404} C_VEL
LIN {X 0,Y 323.916,Z 325.446,A -85,B 0,C 180,E1 -15710.806,E2 -15710.806} C_VEL
LIN {X 0,Y 321.796,Z 335.354,A -85,B 0,C 180,E1 -15712.299,E2 -15712.299} C_VEL
LIN {X 0,Y 319.474,Z 345.657,A -85,B 0,C 180,E1 -15714.189,E2 -15714.189} C_VEL
LIN {X 0,Y 317.188,Z 355.156,A -85,B 0,C 180,E1 -15716.361,E2 -15716.361} C_VEL
LIN {X 0,Y 315.374,Z 362.449,A -85,B 0,C 180,E1 -15718.418,E2 -15718.418} C_VEL
LIN {X 0,Y 313.706,Z 369.377,A -85,B 0,C 180,E1 -15720.882,E2 -15720.882} C_VEL
LIN {X 0,Y 312.494,Z 374.557,A -85,B 0,C 180,E1 -15723.267,E2 -15723.267} C_VEL
LIN {X 0,Y 311.941,Z 376.953,A -85,B 0,C 180,E1 -15724.653,E2 -15724.653} C_VEL
LIN {X 0,Y 311.158,Z 380.508,A -85,B 0,C 180,E1 -15727.418,E2 -15727.418} C_VEL
LIN {X 0,Y 310.893,Z 381.693,A -85,B 0,C 180,E1 -15728.794,E2 -15728.794} C_VEL
LIN {X 0,Y 310.558,Z 382.918,A -85,B 0,C 180,E1 -15731.527,E2 -15731.527} C_VEL
LIN {X 0,Y 310.431,Z 382.708,A -85,B 0,C 180,E1 -15734.234,E2 -15734.234} C_VEL
LIN {X 0,Y 310.571,Z 381.089,A -85,B 0,C 180,E1 -15736.919,E2 -15736.919} C_VEL
LIN {X 0,Y 310.774,Z 378.063,A -85,B 0,C 180,E1 -15739.575,E2 -15739.575} C_VEL
LIN {X 0,Y 311.278,Z 373.557,A -85,B 0,C 180,E1 -15742.213,E2 -15742.213} C_VEL
LIN {X 0,Y 311.754,Z 369.094,A -85,B 0,C 180,E1 -15744.176,E2 -15744.176} C_VEL
LIN {X 0,Y 312.55,Z 362.643,A -85,B 0,C 180,E1 -15746.453,E2 -15746.453} C_VEL
LIN {X 0,Y 313.72,Z 354.626,A -85,B 0,C 180,E1 -15748.715,E2 -15748.715} C_VEL
LIN {X 0,Y 314.95,Z 346.248,A -85,B 0,C 180,E1 -15750.637,E2 -15750.637} C_VEL
LIN {X 0,Y 316.446,Z 336.164,A -85,B 0,C 180,E1 -15752.544,E2 -15752.544} C_VEL
LIN {X 0,Y 317.834,Z 326.031,A -85,B 0,C 180,E1 -15754.119,E2 -15754.119} C_VEL
LIN {X 0,Y 319.485,Z 313.69,A -85,B 0,C 180,E1 -15755.679,E2 -15755.679} C_VEL
LIN {X 0,Y 320.933,Z 301.472,A -85,B 0,C 180,E1 -15756.916,E2 -15756.916} C_VEL
LIN {X 0,Y 322.255,Z 287.931,A -85,B 0,C 180,E1 -15757.99,E2 -15757.99} C_VEL
LIN {X 0,Y 323.282,Z 273.775,A -85,B 0,C 180,E1 -15758.83,E2 -15758.83} C_VEL
LIN {X 0,Y 324.015,Z 259.827,A -85,B 0,C 180,E1 -15759.4,E2 -15759.4} C_VEL
LIN {X 0,Y 324.879,Z 229.947,A -85,B 0,C 180,E1 -15760.102,E2 -15760.102} C_VEL
LIN {X 0,Y 326.793,Z 156.667,A -85,B 0,C 180,E1 -15761.704,E2 -15761.704} C_VEL
LIN {X 0,Y 325.057,Z 150.929,A -85,B 0,C 180,E1 -15761.974,E2 -15761.974} C_VEL
LIN {X 0,Y 316.923,Z 129.752,A -85,B 0,C 180,E1 -15763.14,E2 -15763.14} C_VEL
LIN {X 0,Y 313.682,Z 121.551,A -85,B 0,C 180,E1 -15763.641,E2 -15763.641} C_VEL
LIN {X 0,Y 312.657,Z 117.171,A -85,B 0,C 180,E1 -15765.048,E2 -15765.048} C_VEL
LIN {X 0,Y 312.612,Z 117.172,A -85,B 0,C 180,E1 -15769.245,E2 -15769.245} C_VEL
LIN {X 0,Y 312.557,Z 117.176,A -85,B 0,C 180,E1 -15772.81,E2 -15772.81} C_VEL
LIN {X 0,Y 312.522,Z 117.179,A -85,B 0,C 180,E1 -15776.726,E2 -15776.726} C_VEL
LIN {X 0,Y 312.513,Z 117.181,A -85,B 0,C 180,E1 -15779.651,E2 -15779.651} C_VEL
LIN {X 0,Y 312.48,Z 117.185,A -85,B 0,C 180,E1 -15780.812,E2 -15780.812} C_VEL
LIN {X 0,Y 311.843,Z 117.268,A -85,B 0,C 180,E1 -15781.888,E2 -15781.888} C_VEL
LIN {X 0,Y 309.014,Z 117.618,A -85,B 0,C 180,E1 -15783.639,E2 -15783.639} C_VEL
LIN {X 0,Y 306.603,Z 117.92,A -85,B 0,C 180,E1 -15785.059,E2 -15785.059} C_VEL
LIN {X 0,Y 305.573,Z 118.044,A -85,B 0,C 180,E1 -15786.159,E2 -15786.159} C_VEL
LIN {X 0,Y 305.493,Z 118.055,A -85,B 0,C 180,E1 -15786.531,E2 -15786.531} C_VEL
LIN {X 0,Y 305.498,Z 118.054,A -85,B 0,C 180,E1 -15790.098,E2 -15790.098} C_VEL
LIN {X 0,Y 305.511,Z 118.044,A -85,B 0,C 180,E1 -15793.637,E2 -15793.637} C_VEL
LIN {X 0,Y 305.494,Z 118.054,A -85,B 0,C 180,E1 -15797.403,E2 -15797.403} C_VEL
LIN {X 0,Y 305.493,Z 118.045,A -85,B 0,C 180,E1 -15801.607,E2 -15801.607} C_VEL
LIN {X 0,Y 305.437,Z 118.061,A -85,B 0,C 180,E1 -15804.89,E2 -15804.89} C_VEL
LIN {X 0,Y 305.432,Z 118.063,A -85,B 0,C 180,E1 -15808.357,E2 -15808.357} C_VEL
LIN {X 0,Y 305.497,Z 118.043,A -85,B 0,C 180,E1 -15811.118,E2 -15811.118} C_VEL
LIN {X 0,Y 305.552,Z 118.046,A -85,B 0,C 180,E1 -15814.092,E2 -15814.092} C_VEL
LIN {X 0,Y 305.535,Z 118.049,A -85,B 0,C 180,E1 -15818.411,E2 -15818.411} C_VEL
LIN {X 0,Y 305.582,Z 118.042,A -85,B 0,C 180,E1 -15821.222,E2 -15821.222} C_VEL
LIN {X 0,Y 305.632,Z 118.036,A -85,B 0,C 180,E1 -15825.353,E2 -15825.353} C_VEL
LIN {X 0,Y 305.625,Z 118.04,A -85,B 0,C 180,E1 -15829.404,E2 -15829.404} C_VEL
LIN {X 0,Y 305.798,Z 118.009,A -85,B 0,C 180,E1 -15832.079,E2 -15832.079} C_VEL
LIN {X 0,Y 305.68,Z 118.022,A -85,B 0,C 180,E1 -15834.728,E2 -15834.728} C_VEL
LIN {X 0,Y 305.95,Z 117.997,A -85,B 0,C 180,E1 -15838.688,E2 -15838.688} C_VEL
LIN {X 0,Y 305.949,Z 117.998,A -85,B 0,C 180,E1 -15841.321,E2 -15841.321} C_VEL
LIN {X 0,Y 305.844,Z 118.006,A -85,B 0,C 180,E1 -15846.602,E2 -15846.602} C_VEL
LIN {X 0,Y 305.728,Z 118.028,A -85,B 0,C 180,E1 -15849.264,E2 -15849.264} C_VEL
LIN {X 0,Y 305.583,Z 118.045,A -85,B 0,C 180,E1 -15853.3,E2 -15853.3} C_VEL
LIN {X 0,Y 305.589,Z 118.042,A -85,B 0,C 180,E1 -15856.024,E2 -15856.024} C_VEL
LIN {X 0,Y 305.573,Z 118.045,A -85,B 0,C 180,E1 -15859.449,E2 -15859.449} C_VEL
LIN {X 0,Y 305.487,Z 118.056,A -85,B 0,C 180,E1 -15863.045,E2 -15863.045} C_VEL
LIN {X 0,Y 305.545,Z 118.049,A -85,B 0,C 180,E1 -15866.231,E2 -15866.231} C_VEL
LIN {X 0,Y 305.494,Z 118.053,A -85,B 0,C 180,E1 -15869.054,E2 -15869.054} C_VEL
LIN {X 0,Y 305.464,Z 118.056,A -85,B 0,C 180,E1 -15873.521,E2 -15873.521} C_VEL
LIN {X 0,Y 305.475,Z 118.057,A -85,B 0,C 180,E1 -15876.743,E2 -15876.743} C_VEL
LIN {X 0,Y 305.456,Z 118.057,A -85,B 0,C 180,E1 -15880.603,E2 -15880.603} C_VEL
LIN {X 0,Y 305.427,Z 118.065,A -85,B 0,C 180,E1 -15883.659,E2 -15883.659} C_VEL
LIN {X 0,Y 305.458,Z 118.061,A -85,B 0,C 180,E1 -15887.418,E2 -15887.418} C_VEL
LIN {X 0,Y 305.479,Z 118.058,A -85,B 0,C 180,E1 -15891.601,E2 -15891.601} C_VEL
LIN {X 0,Y 305.493,Z 118.103,A -85,B 0,C 180,E1 -15894.793,E2 -15894.793} C_VEL
LIN {X 0,Y 308.363,Z 130.555,A -85,B 0,C 180,E1 -15898.388,E2 -15898.388} C_VEL
LIN {X 0,Y 309.606,Z 136.525,A -85,B 0,C 180,E1 -15900.042,E2 -15900.042} C_VEL
LIN {X 0,Y 314.854,Z 150.717,A -85,B 0,C 180,E1 -15900.845,E2 -15900.845} C_VEL
LIN {X 0,Y 319.825,Z 182.603,A -85,B 0,C 180,E1 -15902.023,E2 -15902.023} C_VEL
LIN {X 0,Y 317.379,Z 274.684,A -85,B 0,C 180,E1 -15904.112,E2 -15904.112} C_VEL
LIN {X 0,Y 316.505,Z 288.58,A -85,B 0,C 180,E1 -15904.653,E2 -15904.653} C_VEL
LIN {X 0,Y 315.199,Z 302.802,A -85,B 0,C 180,E1 -15905.465,E2 -15905.465} C_VEL
LIN {X 0,Y 313.86,Z 315.762,A -85,B 0,C 180,E1 -15906.471,E2 -15906.471} C_VEL
LIN {X 0,Y 312.34,Z 328.048,A -85,B 0,C 180,E1 -15907.687,E2 -15907.687} C_VEL
LIN {X 0,Y 310.863,Z 338.605,A -85,B 0,C 180,E1 -15908.969,E2 -15908.969} C_VEL
LIN {X 0,Y 309.31,Z 348.558,A -85,B 0,C 180,E1 -15910.421,E2 -15910.421} C_VEL
LIN {X 0,Y 307.929,Z 357.89,A -85,B 0,C 180,E1 -15912.056,E2 -15912.056} C_VEL
LIN {X 0,Y 306.608,Z 367.226,A -85,B 0,C 180,E1 -15914.036,E2 -15914.036} C_VEL
LIN {X 0,Y 305.587,Z 374.987,A -85,B 0,C 180,E1 -15916.028,E2 -15916.028} C_VEL
LIN {X 0,Y 304.737,Z 381.432,A -85,B 0,C 180,E1 -15918.022,E2 -15918.022} C_VEL
LIN {X 0,Y 304.158,Z 386.711,A -85,B 0,C 180,E1 -15920.022,E2 -15920.022} C_VEL
LIN {X 0,Y 303.834,Z 391.01,A -85,B 0,C 180,E1 -15922.024,E2 -15922.024} C_VEL
LIN {X 0,Y 303.608,Z 395.328,A -85,B 0,C 180,E1 -15924.689,E2 -15924.689} C_VEL
LIN {X 0,Y 303.605,Z 398.172,A -85,B 0,C 180,E1 -15927.348,E2 -15927.348} C_VEL
LIN {X 0,Y 303.609,Z 399.622,A -85,B 0,C 180,E1 -15930.002,E2 -15930.002} C_VEL
LIN {X 0,Y 303.6,Z 399.724,A -85,B 0,C 180,E1 -15932.655,E2 -15932.655} C_VEL
LIN {X 0,Y 303.63,Z 398.345,A -85,B 0,C 180,E1 -15935.531,E2 -15935.531} C_VEL
LIN {X 0,Y 303.923,Z 395.935,A -85,B 0,C 180,E1 -15937.977,E2 -15937.977} C_VEL
LIN {X 0,Y 304.548,Z 391.957,A -85,B 0,C 180,E1 -15940.64,E2 -15940.64} C_VEL
LIN {X 0,Y 305.705,Z 386.446,A -85,B 0,C 180,E1 -15943.293,E2 -15943.293} C_VEL
LIN {X 0,Y 307.378,Z 379.254,A -85,B 0,C 180,E1 -15945.926,E2 -15945.926} C_VEL
LIN {X 0,Y 309.198,Z 371.359,A -85,B 0,C 180,E1 -15948.214,E2 -15948.214} C_VEL
LIN {X 0,Y 311.239,Z 363.142,A -85,B 0,C 180,E1 -15950.144,E2 -15950.144} C_VEL
LIN {X 0,Y 313.658,Z 353.279,A -85,B 0,C 180,E1 -15952.045,E2 -15952.045} C_VEL
LIN {X 0,Y 316.195,Z 342.349,A -85,B 0,C 180,E1 -15953.759,E2 -15953.759} C_VEL
LIN {X 0,Y 318.717,Z 330.225,A -85,B 0,C 180,E1 -15955.294,E2 -15955.294} C_VEL
LIN {X 0,Y 320.955,Z 318.26,A -85,B 0,C 180,E1 -15956.499,E2 -15956.499} C_VEL
LIN {X 0,Y 322.93,Z 305.082,A -85,B 0,C 180,E1 -15957.548,E2 -15957.548} C_VEL
LIN {X 0,Y 324.752,Z 291.41,A -85,B 0,C 180,E1 -15958.345,E2 -15958.345} C_VEL
LIN {X 0,Y 326.112,Z 277.293,A -85,B 0,C 180,E1 -15958.919,E2 -15958.919} C_VEL
LIN {X 0,Y 326.966,Z 258.096,A -85,B 0,C 180,E1 -15959.409,E2 -15959.409} C_VEL
LIN {X 0,Y 329.569,Z 186.083,A -85,B 0,C 180,E1 -15961.006,E2 -15961.006} C_VEL
LIN {X 0,Y 326.017,Z 166.699,A -85,B 0,C 180,E1 -15961.986,E2 -15961.986} C_VEL
LIN {X 0,Y 319.455,Z 152.538,A -85,B 0,C 180,E1 -15963.276,E2 -15963.276} C_VEL
LIN {X 0,Y 312.241,Z 139.041,A -85,B 0,C 180,E1 -15964.729,E2 -15964.729} C_VEL
LIN {X 0,Y 310.469,Z 135.371,A -85,B 0,C 180,E1 -15965.142,E2 -15965.142} C_VEL
LIN {X 0,Y 307.448,Z 124.64,A -85,B 0,C 180,E1 -15968.99,E2 -15968.99} C_VEL
LIN {X 0,Y 305.435,Z 118.058,A -85,B 0,C 180,E1 -15971.602,E2 -15971.602} C_VEL
LIN {X 0,Y 305.416,Z 118.064,A -85,B 0,C 180,E1 -15975.51,E2 -15975.51} C_VEL
LIN {X 0,Y 305.469,Z 118.037,A -85,B 0,C 180,E1 -15979.4,E2 -15979.4} C_VEL
LIN {X 0,Y 305.469,Z 118.054,A -85,B 0,C 180,E1 -15983.256,E2 -15983.256} C_VEL
LIN {X 0,Y 305.48,Z 118.055,A -85,B 0,C 180,E1 -15986.481,E2 -15986.481} C_VEL
LIN {X 0,Y 305.445,Z 118.058,A -85,B 0,C 180,E1 -15989.585,E2 -15989.585} C_VEL
LIN {X 0,Y 305.473,Z 118.05,A -85,B 0,C 180,E1 -15992.6,E2 -15992.6} C_VEL
LIN {X 0,Y 305.49,Z 118.048,A -85,B 0,C 180,E1 -15995.533,E2 -15995.533} C_VEL
LIN {X 0,Y 305.52,Z 118.042,A -85,B 0,C 180,E1 -15999.811,E2 -15999.811} C_VEL
LIN {X 0,Y 305.588,Z 118.043,A -85,B 0,C 180,E1 -16002.6,E2 -16002.6} C_VEL
LIN {X 0,Y 305.663,Z 118.034,A -85,B 0,C 180,E1 -16005.346,E2 -16005.346} C_VEL
LIN {X 0,Y 305.636,Z 118.036,A -85,B 0,C 180,E1 -16009.396,E2 -16009.396} C_VEL
LIN {X 0,Y 305.757,Z 118.015,A -85,B 0,C 180,E1 -16012.069,E2 -16012.069} C_VEL
LIN {X 0,Y 305.676,Z 118.035,A -85,B 0,C 180,E1 -16014.719,E2 -16014.719} C_VEL
LIN {X 0,Y 305.959,Z 118,A -85,B 0,C 180,E1 -16018.68,E2 -16018.68} C_VEL
LIN {X 0,Y 305.959,Z 117.986,A -85,B 0,C 180,E1 -16021.312,E2 -16021.312} C_VEL
LIN {X 0,Y 305.676,Z 118.023,A -85,B 0,C 180,E1 -16025.272,E2 -16025.272} C_VEL
LIN {X 0,Y 305.769,Z 118.021,A -85,B 0,C 180,E1 -16027.922,E2 -16027.922} C_VEL
LIN {X 0,Y 305.602,Z 118.041,A -85,B 0,C 180,E1 -16031.94,E2 -16031.94} C_VEL
LIN {X 0,Y 305.64,Z 118.039,A -85,B 0,C 180,E1 -16035.03,E2 -16035.03} C_VEL
LIN {X 0,Y 305.576,Z 118.042,A -85,B 0,C 180,E1 -16039.439,E2 -16039.439} C_VEL
LIN {X 0,Y 305.486,Z 118.052,A -85,B 0,C 180,E1 -16043.035,E2 -16043.035} C_VEL
LIN {X 0,Y 305.518,Z 118.047,A -85,B 0,C 180,E1 -16046.212,E2 -16046.212} C_VEL
LIN {X 0,Y 305.465,Z 118.042,A -85,B 0,C 180,E1 -16049.036,E2 -16049.036} C_VEL
LIN {X 0,Y 305.428,Z 118.066,A -85,B 0,C 180,E1 -16051.948,E2 -16051.948} C_VEL
LIN {X 0,Y 305.476,Z 118.063,A -85,B 0,C 180,E1 -16056.053,E2 -16056.053} C_VEL
LIN {X 0,Y 305.494,Z 118.118,A -85,B 0,C 180,E1 -16056.369,E2 -16056.369} C_VEL
LIN {X 0,Y 306.884,Z 123.09,A -85,B 0,C 180,E1 -16058.363,E2 -16058.363} C_VEL
LIN {X 0,Y 309.458,Z 127.357,A -85,B 0,C 180,E1 -16058.91,E2 -16058.91} C_VEL
LIN {X 0,Y 316.937,Z 140.175,A -85,B 0,C 180,E1 -16060.43,E2 -16060.43} C_VEL
LIN {X 0,Y 324.663,Z 155.076,A -85,B 0,C 180,E1 -16061.936,E2 -16061.936} C_VEL
LIN {X 0,Y 330.183,Z 166.909,A -85,B 0,C 180,E1 -16062.981,E2 -16062.981} C_VEL
LIN {X 0,Y 326.787,Z 259.033,A -85,B 0,C 180,E1 -16065.055,E2 -16065.055} C_VEL
LIN {X 0,Y 325.627,Z 273.682,A -85,B 0,C 180,E1 -16065.622,E2 -16065.622} C_VEL
LIN {X 0,Y 324.122,Z 287.132,A -85,B 0,C 180,E1 -16066.384,E2 -16066.384} C_VEL
LIN {X 0,Y 322.234,Z 301.006,A -85,B 0,C 180,E1 -16067.457,E2 -16067.457} C_VEL
LIN {X 0,Y 320.265,Z 312.46,A -85,B 0,C 180,E1 -16068.581,E2 -16068.581} C_VEL
LIN {X 0,Y 317.768,Z 324.915,A -85,B 0,C 180,E1 -16070.103,E2 -16070.103} C_VEL
LIN {X 0,Y 315.318,Z 335.987,A -85,B 0,C 180,E1 -16071.791,E2 -16071.791} C_VEL
LIN {X 0,Y 313.152,Z 345.154,A -85,B 0,C 180,E1 -16073.505,E2 -16073.505} C_VEL
LIN {X 0,Y 310.869,Z 354.292,A -85,B 0,C 180,E1 -16075.583,E2 -16075.583} C_VEL
LIN {X 0,Y 308.787,Z 362.143,A -85,B 0,C 180,E1 -16077.794,E2 -16077.794} C_VEL
LIN {X 0,Y 307.325,Z 367.88,A -85,B 0,C 180,E1 -16079.793,E2 -16079.793} C_VEL
LIN {X 0,Y 306.053,Z 372.81,A -85,B 0,C 180,E1 -16081.915,E2 -16081.915} C_VEL
LIN {X 0,Y 305.094,Z 376.699,A -85,B 0,C 180,E1 -16084.042,E2 -16084.042} C_VEL
LIN {X 0,Y 304.189,Z 380.401,A -85,B 0,C 180,E1 -16086.871,E2 -16086.871} C_VEL
LIN {X 0,Y 303.63,Z 382.551,A -85,B 0,C 180,E1 -16089.682,E2 -16089.682} C_VEL
LIN {X 0,Y 303.405,Z 383.222,A -85,B 0,C 180,E1 -16092.473,E2 -16092.473} C_VEL
LIN {X 0,Y 303.375,Z 382.44,A -85,B 0,C 180,E1 -16095.235,E2 -16095.235} C_VEL
LIN {X 0,Y 303.464,Z 381.519,A -85,B 0,C 180,E1 -16096.607,E2 -16096.607} C_VEL
LIN {X 0,Y 303.641,Z 378.627,A -85,B 0,C 180,E1 -16099.327,E2 -16099.327} C_VEL
LIN {X 0,Y 304.022,Z 375.52,A -85,B 0,C 180,E1 -16101.356,E2 -16101.356} C_VEL
LIN {X 0,Y 304.63,Z 369.942,A -85,B 0,C 180,E1 -16104.039,E2 -16104.039} C_VEL
LIN {X 0,Y 305.409,Z 363.653,A -85,B 0,C 180,E1 -16106.37,E2 -16106.37} C_VEL
LIN {X 0,Y 306.568,Z 355.816,A -85,B 0,C 180,E1 -16108.685,E2 -16108.685} C_VEL
LIN {X 0,Y 307.831,Z 347.637,A -85,B 0,C 180,E1 -16110.652,E2 -16110.652} C_VEL
LIN {X 0,Y 309.356,Z 337.786,A -85,B 0,C 180,E1 -16112.602,E2 -16112.602} C_VEL
LIN {X 0,Y 310.907,Z 326.871,A -85,B 0,C 180,E1 -16114.374,E2 -16114.374} C_VEL
LIN {X 0,Y 312.605,Z 314.728,A -85,B 0,C 180,E1 -16115.966,E2 -16115.966} C_VEL
LIN {X 0,Y 314.108,Z 302.717,A -85,B 0,C 180,E1 -16117.228,E2 -16117.228} C_VEL
LIN {X 0,Y 315.399,Z 289.509,A -85,B 0,C 180,E1 -16118.326,E2 -16118.326} C_VEL
LIN {X 0,Y 316.54,Z 275.773,A -85,B 0,C 180,E1 -16119.181,E2 -16119.181} C_VEL
LIN {X 0,Y 317.315,Z 261.62,A -85,B 0,C 180,E1 -16119.801,E2 -16119.801} C_VEL
LIN {X 0,Y 318.011,Z 241.203,A -85,B 0,C 180,E1 -16120.323,E2 -16120.323} C_VEL
LIN {X 0,Y 320.293,Z 157.684,A -85,B 0,C 180,E1 -16122.183,E2 -16122.183} C_VEL
LIN {X 0,Y 312.493,Z 136.548,A -85,B 0,C 180,E1 -16123.34,E2 -16123.34} C_VEL
LIN {X 0,Y 306.459,Z 121.749,A -85,B 0,C 180,E1 -16124.271,E2 -16124.271} C_VEL
LIN {X 0,Y 305.606,Z 118.05,A -85,B 0,C 180,E1 -16125.505,E2 -16125.505} C_VEL
LIN {X 0,Y 305.58,Z 118.049,A -85,B 0,C 180,E1 -16129.465,E2 -16129.465} C_VEL
LIN {X 0,Y 305.521,Z 118.054,A -85,B 0,C 180,E1 -16133.071,E2 -16133.071} C_VEL
LIN {X 0,Y 305.515,Z 118.051,A -85,B 0,C 180,E1 -16136.228,E2 -16136.228} C_VEL
